KUKA KRL program: MyProgram_234().src

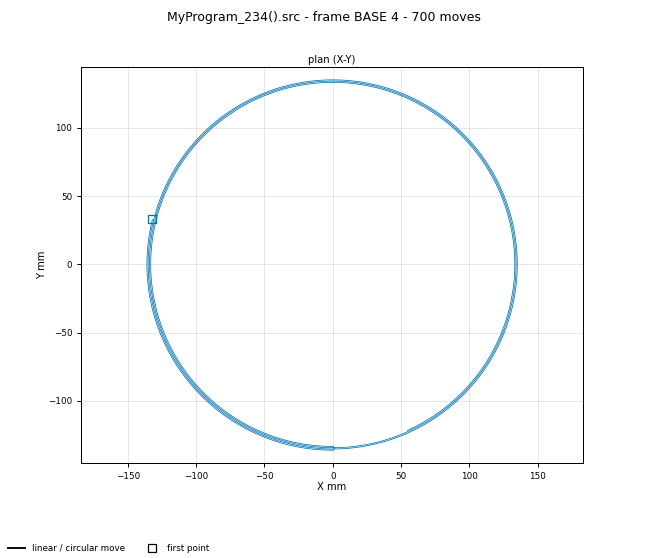
[picture p0: tool path of MyProgram_234().src in frame BASE 4, 700 of 700 moves have a stored position in this frame; points joined in program order, loops and branches not executed]
&ACCESS RVP
&REL 1
&PARAM TEMPLATE = C:\KRC\Roboter\Template\vorgabe
&PARAM EDITMASK = *
DEF MyProgram_234()
; ---- Setting reference (Base) ----
$BASE = BASE_DATA[4]

; --------------------------
; ---- Setting tool (TCP) ----
$TOOL = TOOL_DATA[3]
; --------------------------

$VEL.CP = VEL_APROX_PRINT
Startdeposition()
$VEL.CP = VEL_PRINT
LIN {X -132.079,Y 32.9632,Z 159,A 163.3178,B 23.9128,C -1.2869,E1 23.7896,E2 283.5753} C_DIS
LIN {X -133.2514,Y 27.8523,Z 159,A 165.544,B 23.9131,C -1.2806,E1 23.7882,E2 281.3509} C_DIS
LIN {X -134.047,Y 23.7201,Z 159,A 167.2359,B 23.9136,C -1.2711,E1 23.7874,E2 279.6721} C_DIS
LIN {X -134.6969,Y 19.7013,Z 159,A 168.9686,B 23.9138,C -1.2664,E1 23.7867,E2 277.9401} C_DIS
LIN {X -135.173,Y 16.1077,Z 159,A 170.4984,B 23.914,C -1.2616,E1 23.7861,E2 276.4127} C_DIS
LIN {X -135.6084,Y 11.907,Z 159,A 172.2964,B 23.9143,C -1.2567,E1 23.7857,E2 274.6154} C_DIS
LIN {X -135.8889,Y 8.0937,Z 159,A 173.8881,B 23.9146,C -1.2506,E1 23.7854,E2 273.0289} C_DIS
LIN {X -136.071,Y 3.9947,Z 159,A 175.6367,B 23.9148,C -1.246,E1 23.7852,E2 271.2807} C_DIS
LIN {X -136.1316,Y 0.0516,Z 159,A 177.3098,B 23.9151,C -1.2411,E1 23.7852,E2 269.609} C_DIS
LIN {X -136.08,Y -3.6704,Z 159,A 178.9234,B 23.9151,C -1.2383,E1 23.7852,E2 267.9922} C_DIS
LIN {X -135.9057,Y -7.8204,Z 159,A -179.3031,B 23.9154,C -1.2338,E1 23.7855,E2 266.2187} C_DIS
LIN {X -135.6203,Y -11.7657,Z 159,A -177.6067,B 23.9156,C -1.2299,E1 23.7859,E2 264.5213} C_DIS
LIN {X -135.25,Y -15.4619,Z 159,A -176.0236,B 23.9158,C -1.2258,E1 23.7863,E2 262.9385} C_DIS
LIN {X -134.7524,Y -19.3124,Z 159,A -174.416,B 23.9161,C -1.2192,E1 23.787,E2 261.337} C_DIS
LIN {X -133.9612,Y -24.1999,Z 159,A -171.5444,B 23.9146,C -1.2507,E1 23.7884,E2 258.3695} C_DIS
LIN {X -132.7292,Y -30.2346,Z 159,A -169.7414,B 23.9168,C -1.2043,E1 23.7894,E2 256.6705} C_DIS
LIN {X -131.8389,Y -33.9095,Z 159,A -168.2744,B 23.9173,C -1.1933,E1 23.7904,E2 255.2218} C_DIS
LIN {X -130.8523,Y -37.5362,Z 159,A -166.5488,B 23.9173,C -1.1953,E1 23.7917,E2 253.4807} C_DIS
LIN {X -129.8374,Y -40.9106,Z 159,A -165.065,B 23.9175,C -1.1908,E1 23.7929,E2 251.9992} C_DIS
LIN {X -128.7798,Y -44.1262,Z 159,A -163.6167,B 23.9176,C -1.1876,E1 23.7942,E2 250.5501} C_DIS
LIN {X -127.6866,Y -47.1974,Z 159,A -162.2254,B 23.9178,C -1.1844,E1 23.7955,E2 249.1585} C_DIS
LIN {X -126.4518,Y -50.4114,Z 159,A -160.7598,B 23.9179,C -1.1808,E1 23.797,E2 247.693} C_DIS
LIN {X -125.049,Y -53.7951,Z 159,A -159.4632,B 23.9187,C -1.1645,E1 23.7984,E2 246.4294} C_DIS
LIN {X -123.7178,Y -56.7903,Z 159,A -157.1398,B 23.9167,C -1.2064,E1 23.8013,E2 243.9887} C_DIS
LIN {X -121.2923,Y -61.8002,Z 159,A -155.5783,B 23.9188,C -1.1616,E1 23.8031,E2 242.5295} C_DIS
LIN {X -119.8894,Y -64.4838,Z 159,A -154.1181,B 23.9186,C -1.167,E1 23.805,E2 241.0477} C_DIS
LIN {X -117.6694,Y -68.4517,Z 159,A -152.2675,B 23.9189,C -1.1587,E1 23.8076,E2 239.2075} C_DIS
LIN {X -115.4192,Y -72.1811,Z 159,A -150.4067,B 23.9191,C -1.1551,E1 23.8103,E2 237.3456} C_DIS
LIN {X -113.1889,Y -75.6301,Z 159,A -148.648,B 23.9192,C -1.1521,E1 23.813,E2 235.5853} C_DIS
LIN {X -110.6731,Y -79.266,Z 159,A -146.7601,B 23.9194,C -1.1486,E1 23.816,E2 233.6961} C_DIS
LIN {X -107.9492,Y -82.9378,Z 159,A -144.8663,B 23.9197,C -1.1423,E1 23.8192,E2 231.8084} C_DIS
LIN {X -105.2261,Y -86.3665,Z 159,A -143.017,B 23.9199,C -1.1382,E1 23.8224,E2 229.9603} C_DIS
LIN {X -101.84,Y -90.3343,Z 159,A -140.897,B 23.9203,C -1.1294,E1 23.8263,E2 227.8521} C_DIS
LIN {X -99.3816,Y -93.0324,Z 159,A -139.2141,B 23.9201,C -1.1331,E1 23.8295,E2 226.1522} C_DIS
LIN {X -96.907,Y -95.6073,Z 159,A -137.545,B 23.9199,C -1.138,E1 23.8328,E2 224.4634} C_DIS
LIN {X -92.9629,Y -99.4464,Z 159,A -135.351,B 23.9204,C -1.127,E1 23.8372,E2 222.287} C_DIS
LIN {X -89.9747,Y -102.157,Z 159,A -133.0559,B 23.9192,C -1.1534,E1 23.8422,E2 219.9171} C_DIS
LIN {X -85.7356,Y -105.741,Z 159,A -131.3189,B 23.9207,C -1.1189,E1 23.8458,E2 218.2586} C_DIS
LIN {X -82.7538,Y -108.0899,Z 159,A -129.715,B 23.9208,C -1.1163,E1 23.8493,E2 216.655} C_DIS
LIN {X -79.0794,Y -110.8065,Z 159,A -127.8281,B 23.9211,C -1.1111,E1 23.8535,E2 214.774} C_DIS
LIN {X -75.5469,Y -113.2444,Z 159,A -126.0361,B 23.9212,C -1.1074,E1 23.8577,E2 212.9849} C_DIS
LIN {X -72.6974,Y -115.0944,Z 159,A -124.2034,B 23.9204,C -1.1254,E1 23.8621,E2 211.1015} C_DIS
LIN {X -69.2355,Y -117.21,Z 159,A -122.8138,B 23.9213,C -1.1068,E1 23.8654,E2 209.7535} C_DIS
LIN {X -66.0235,Y -119.0485,Z 159,A -121.2797,B 23.9214,C -1.1035,E1 23.8691,E2 208.223} C_DIS
LIN {X -62.1027,Y -121.1383,Z 159,A -119.4931,B 23.9217,C -1.0968,E1 23.8735,E2 206.4477} C_DIS
LIN {X -59.0691,Y -122.6463,Z 159,A -118.0743,B 23.9217,C -1.0947,E1 23.877,E2 205.0303} C_DIS
LIN {X -52.286,Y -125.6874,Z 159,A -114.8574,B 23.9217,C -1.0956,E1 23.8853,E2 201.8031} C_DIS
LIN {X -47.9859,Y -127.3913,Z 159,A -112.8439,B 23.9217,C -1.097,E1 23.8905,E2 199.7815} C_DIS
LIN {X -43.4345,Y -129.0146,Z 159,A -110.8603,B 23.9219,C -1.0927,E1 23.8958,E2 197.8045} C_DIS
LIN {X -39.8208,Y -130.1746,Z 159,A -109.3213,B 23.922,C -1.0885,E1 23.8998,E2 196.273} C_DIS
LIN {X -36.6839,Y -131.0932,Z 159,A -107.9375,B 23.922,C -1.088,E1 23.9036,E2 194.8882} C_DIS
LIN {X -32.9741,Y -132.0762,Z 159,A -106.2345,B 23.922,C -1.0915,E1 23.9082,E2 193.174} C_DIS
LIN {X -28.9465,Y -133.0162,Z 159,A -104.5737,B 23.9221,C -1.0865,E1 23.9127,E2 191.5233} C_DIS
LIN {X -25.5638,Y -133.7074,Z 159,A -103.1858,B 23.9223,C -1.0826,E1 23.9165,E2 190.1435} C_DIS
LIN {X -20.5942,Y -134.5627,Z 159,A -100.9853,B 23.9222,C -1.0859,E1 23.9226,E2 187.9326} C_DIS
LIN {X -16.4484,Y -135.1324,Z 159,A -98.8515,B 23.9213,C -1.1049,E1 23.9286,E2 185.7503} C_DIS
LIN {X -12.5936,Y -135.5462,Z 159,A -96.9315,B 23.9207,C -1.1198,E1 23.9341,E2 183.7925} C_DIS
LIN {X -7.2101,Y -135.9389,Z 159,A -95.2727,B 23.9221,C -1.0878,E1 23.9385,E2 182.212} C_DIS
LIN {X 0.5173,Y -136.1287,Z 159,A -91.6014,B 23.9211,C -1.1103,E1 23.9489,E2 178.4853} C_DIS
LIN {X 0.5173,Y -136.1287,Z 159,A -91.6014,B 23.9211,C -1.1103,E1 23.9489,E2 178.4853} C_DIS
Enddeposition()
LIN {X 0.9368,Y -135.1941,Z 159,A -91.8649,B 22.4196,C -0.8172,E1 22.4349,E2 179.316} C_DIS
Startdeposition()
$VEL.CP = VEL_PRINT
LIN {X -3.0281,Y -135.1695,Z 159,A -93.7042,B 22.4199,C -0.8092,E1 22.4297,E2 181.1764} C_DIS
LIN {X -7.7949,Y -134.9776,Z 159,A -95.9195,B 22.4202,C -0.7999,E1 22.4234,E2 183.4167} C_DIS
LIN {X -13.0956,Y -134.5658,Z 159,A -98.0516,B 22.42,C -0.8058,E1 22.4175,E2 185.5345} C_DIS
LIN {X -16.1305,Y -134.2357,Z 159,A -99.3289,B 22.42,C -0.8068,E1 22.414,E2 186.8101} C_DIS
LIN {X -19.4901,Y -133.7897,Z 159,A -100.8591,B 22.42,C -0.8027,E1 22.4097,E2 188.3524} C_DIS
LIN {X -23.6224,Y -133.1218,Z 159,A -102.3216,B 22.4196,C -0.8179,E1 22.4058,E2 189.7764} C_DIS
LIN {X -26.7677,Y -132.5251,Z 159,A -103.9188,B 22.4199,C -0.8072,E1 22.4014,E2 191.4039} C_DIS
LIN {X -30.2748,Y -131.7681,Z 159,A -105.4244,B 22.4199,C -0.8086,E1 22.3973,E2 192.9078} C_DIS
LIN {X -33.5797,Y -130.9652,Z 159,A -106.8089,B 22.4198,C -0.8121,E1 22.3935,E2 194.2854} C_DIS
LIN {X -36.6063,Y -130.1514,Z 159,A -108.1864,B 22.4198,C -0.8107,E1 22.3898,E2 195.669} C_DIS
LIN {X -39.882,Y -129.1855,Z 159,A -109.6302,B 22.4198,C -0.8119,E1 22.3859,E2 197.1124} C_DIS
LIN {X -43.3138,Y -128.0767,Z 159,A -111.3197,B 22.42,C -0.8056,E1 22.3814,E2 198.8218} C_DIS
LIN {X -47.6534,Y -126.5249,Z 159,A -113.1109,B 22.4197,C -0.8149,E1 22.3768,E2 200.5927} C_DIS
LIN {X -50.6546,Y -125.3533,Z 159,A -114.5476,B 22.4197,C -0.813,E1 22.373,E2 202.038} C_DIS
LIN {X -54.6129,Y -123.6817,Z 159,A -116.7429,B 22.4203,C -0.7977,E1 22.3673,E2 204.2792} C_DIS
LIN {X -58.0744,Y -122.0931,Z 159,A -117.7099,B 22.4192,C -0.8294,E1 22.365,E2 205.1657} C_DIS
LIN {X -62.044,Y -120.1269,Z 159,A -119.8272,B 22.4195,C -0.8207,E1 22.3597,E2 207.3123} C_DIS
LIN {X -64.6397,Y -118.75,Z 159,A -121.1817,B 22.4195,C -0.8173,E1 22.3563,E2 208.6799} C_DIS
LIN {X -68.3399,Y -116.6599,Z 159,A -123.4642,B 22.4203,C -0.798,E1 22.3507,E2 211.0209} C_DIS
LIN {X -72.4236,Y -114.1698,Z 159,A -124.6995,B 22.4189,C -0.8371,E1 22.348,E2 212.1577} C_DIS
LIN {X -76.606,Y -111.4063,Z 159,A -127.1393,B 22.4193,C -0.8262,E1 22.3422,E2 214.6355} C_DIS
LIN {X -80.2636,Y -108.801,Z 159,A -129.009,B 22.4191,C -0.831,E1 22.338,E2 216.4999} C_DIS
LIN {X -83.739,Y -106.1494,Z 159,A -130.9102,B 22.4191,C -0.8321,E1 22.3338,E2 218.4059} C_DIS
LIN {X -87.1969,Y -103.3281,Z 159,A -133.1146,B 22.4194,C -0.8216,E1 22.329,E2 220.6475} C_DIS
LIN {X -90.0311,Y -100.8676,Z 159,A -134.0842,B 22.4183,C -0.8528,E1 22.3271,E2 221.5394} C_DIS
LIN {X -93.7404,Y -97.4307,Z 159,A -136.5561,B 22.4187,C -0.8423,E1 22.322,E2 224.0503} C_DIS
LIN {X -96.7962,Y -94.3953,Z 159,A -138.4289,B 22.4187,C -0.8441,E1 22.3183,E2 225.9274} C_DIS
LIN {X -99.8464,Y -91.1631,Z 159,A -140.1658,B 22.4183,C -0.8548,E1 22.315,E2 227.6446} C_DIS
LIN {X -102.1643,Y -88.5577,Z 159,A -141.8369,B 22.4185,C -0.8496,E1 22.3119,E2 229.338} C_DIS
LIN {X -105.1304,Y -85.0145,Z 159,A -143.761,B 22.4182,C -0.8557,E1 22.3085,E2 231.256} C_DIS
LIN {X -108.0038,Y -81.3329,Z 159,A -145.7259,B 22.418,C -0.8612,E1 22.3052,E2 233.217} C_DIS
LIN {X -110.675,Y -77.6594,Z 159,A -147.7071,B 22.418,C -0.8635,E1 22.3019,E2 235.2031} C_DIS
LIN {X -113.2164,Y -73.9053,Z 159,A -149.6464,B 22.4178,C -0.8677,E1 22.2989,E2 237.1425} C_DIS
LIN {X -115.5116,Y -70.2641,Z 159,A -151.4667,B 22.4176,C -0.8726,E1 22.2963,E2 238.9601} C_DIS
LIN {X -117.7755,Y -66.3988,Z 159,A -153.3603,B 22.4174,C -0.878,E1 22.2936,E2 240.8508} C_DIS
LIN {X -119.7044,Y -62.8503,Z 159,A -155.0786,B 22.4173,C -0.8824,E1 22.2914,E2 242.5677} C_DIS
LIN {X -121.6017,Y -59.1012,Z 159,A -156.7614,B 22.4169,C -0.8917,E1 22.2893,E2 244.2362} C_DIS
LIN {X -123.8092,Y -54.3244,Z 159,A -158.9741,B 22.4166,C -0.8988,E1 22.2868,E2 246.4438} C_DIS
LIN {X -124.9315,Y -51.688,Z 159,A -160.3608,B 22.4168,C -0.8947,E1 22.2852,E2 247.8499} C_DIS
LIN {X -126.5688,Y -47.5361,Z 159,A -162.2011,B 22.4165,C -0.9026,E1 22.2834,E2 249.6814} C_DIS
LIN {X -127.8142,Y -44.0784,Z 159,A -163.722,B 22.4163,C -0.9088,E1 22.282,E2 251.1955} C_DIS
LIN {X -129.0675,Y -40.2673,Z 159,A -165.3832,B 22.416,C -0.9156,E1 22.2806,E2 252.8496} C_DIS
LIN {X -130.0053,Y -37.1251,Z 159,A -167.1173,B 22.4164,C -0.9048,E1 22.2792,E2 254.6235} C_DIS
LIN {X -130.8711,Y -33.9505,Z 159,A -168.4639,B 22.4162,C -0.9111,E1 22.2783,E2 255.9622} C_DIS
LIN {X -133.1369,Y -23.5378,Z 159,A -172.7695,B 22.4153,C -0.9344,E1 22.2758,E2 260.2352} C_DIS
LIN {X -133.6941,Y -20.1397,Z 159,A -174.3597,B 22.4153,C -0.9332,E1 22.2751,E2 261.8391} C_DIS
LIN {X -134.2618,Y -15.912,Z 159,A -176.0343,B 22.4148,C -0.9448,E1 22.2745,E2 263.4945} C_DIS
LIN {X -134.6144,Y -12.5897,Z 159,A -177.5154,B 22.4148,C -0.9465,E1 22.2741,E2 264.9812} C_DIS
LIN {X -134.9389,Y -8.4233,Z 159,A -179.2792,B 22.4145,C -0.9524,E1 22.2738,E2 266.7412} C_DIS
LIN {X -135.11,Y -4.9807,Z 159,A 179.14,B 22.4145,C -0.9519,E1 22.2736,E2 268.3341} C_DIS
LIN {X -135.1996,Y -0.8442,Z 159,A 177.4322,B 22.4142,C -0.9595,E1 22.2736,E2 270.0335} C_DIS
LIN {X -135.1606,Y 3.3519,Z 159,A 175.6326,B 22.4141,C -0.9643,E1 22.2736,E2 271.8327} C_DIS
LIN {X -135.0229,Y 6.949,Z 159,A 174.1184,B 22.4138,C -0.9698,E1 22.2738,E2 273.3427} C_DIS
LIN {X -134.735,Y 11.2223,Z 159,A 172.2572,B 22.4137,C -0.9736,E1 22.2742,E2 275.2065} C_DIS
LIN {X -134.2965,Y 15.6212,Z 159,A 170.3647,B 22.4135,C -0.9788,E1 22.2747,E2 277.0981} C_DIS
LIN {X -133.7907,Y 19.4832,Z 159,A 168.7199,B 22.4132,C -0.9844,E1 22.2754,E2 278.7393} C_DIS
LIN {X -133.0853,Y 23.8263,Z 159,A 166.925,B 22.4128,C -0.9934,E1 22.2762,E2 280.5223} C_DIS
LIN {X -132.4612,Y 27.0816,Z 159,A 165.4622,B 22.4128,C -0.9954,E1 22.277,E2 281.9897} C_DIS
LIN {X -131.5133,Y 31.3644,Z 159,A 163.8004,B 22.4121,C -1.0099,E1 22.278,E2 283.6244} C_DIS
LIN {X -130.7732,Y 34.3223,Z 159,A 161.9635,B 22.413,C -0.9903,E1 22.2793,E2 285.525} C_DIS
LIN {X -129.8613,Y 37.6236,Z 159,A 161.0027,B 22.4119,C -1.0162,E1 22.28,E2 286.4239} C_DIS
LIN {X -128.0076,Y 43.5208,Z 159,A 158.2134,B 22.4119,C -1.0169,E1 22.2824,E2 289.2292} C_DIS
LIN {X -126.5522,Y 47.5804,Z 159,A 156.3461,B 22.4117,C -1.0209,E1 22.2842,E2 291.098} C_DIS
LIN {X -125.2287,Y 50.9637,Z 159,A 154.8328,B 22.4114,C -1.0267,E1 22.2857,E2 292.6055} C_DIS
LIN {X -123.992,Y 53.9014,Z 159,A 153.4528,B 22.4113,C -1.0295,E1 22.2872,E2 293.9866} C_DIS
LIN {X -122.6155,Y 56.9631,Z 159,A 152.0207,B 22.4111,C -1.0334,E1 22.2889,E2 295.4174} C_DIS
LIN {X -121.1128,Y 60.0924,Z 159,A 150.5165,B 22.4111,C -1.0363,E1 22.2907,E2 296.9231} C_DIS
LIN {X -119.2292,Y 63.752,Z 159,A 148.7776,B 22.4108,C -1.0417,E1 22.293,E2 298.6583} C_DIS
LIN {X -117.2847,Y 67.2624,Z 159,A 146.9782,B 22.4108,C -1.0423,E1 22.2955,E2 300.4667} C_DIS
LIN {X -115.0045,Y 71.0913,Z 159,A 145.0611,B 22.4106,C -1.0464,E1 22.2982,E2 302.3841} C_DIS
LIN {X -112.9386,Y 74.3283,Z 159,A 143.4277,B 22.4104,C -1.0507,E1 22.3007,E2 304.0154} C_DIS
LIN {X -110.4125,Y 78.0316,Z 159,A 141.5521,B 22.4101,C -1.057,E1 22.3037,E2 305.885} C_DIS
LIN {X -107.8054,Y 81.5957,Z 159,A 139.556,B 22.4101,C -1.0566,E1 22.307,E2 307.893} C_DIS
LIN {X -105.1746,Y 84.9597,Z 159,A 137.7114,B 22.41,C -1.0598,E1 22.3103,E2 309.7389} C_DIS
LIN {X -99.9633,Y 91.0343,Z 159,A 134.2089,B 22.4098,C -1.0636,E1 22.3167,E2 313.2494} C_DIS
LIN {X -96.201,Y 95.002,Z 159,A 132.0334,B 22.4093,C -1.0754,E1 22.3209,E2 315.4042} C_DIS
LIN {X -92.9702,Y 98.1654,Z 159,A 130.1303,B 22.409,C -1.0805,E1 22.3247,E2 317.3027} C_DIS
LIN {X -89.188,Y 101.6136,Z 159,A 128.0456,B 22.4086,C -1.0892,E1 22.329,E2 319.3739} C_DIS
LIN {X -86.0424,Y 104.291,Z 159,A 125.762,B 22.4095,C -1.0695,E1 22.3341,E2 321.7192} C_DIS
LIN {X -82.4871,Y 107.1256,Z 159,A 123.8971,B 22.4092,C -1.0763,E1 22.3382,E2 323.5739} C_DIS
LIN {X -79.195,Y 109.5811,Z 159,A 122.5954,B 22.4082,C -1.0993,E1 22.341,E2 324.8203} C_DIS
LIN {X -75.9198,Y 111.8751,Z 159,A 120.835,B 22.4082,C -1.0997,E1 22.345,E2 326.5864} C_DIS
LIN {X -69.1781,Y 116.1647,Z 159,A 117.6362,B 22.4075,C -1.1144,E1 22.3525,E2 329.758} C_DIS
LIN {X -66.4481,Y 117.7478,Z 159,A 116.055,B 22.4079,C -1.1058,E1 22.3564,E2 331.3671} C_DIS
LIN {X -62.7463,Y 119.759,Z 159,A 114.3724,B 22.4075,C -1.1134,E1 22.3605,E2 333.0349} C_DIS
LIN {X -59.6838,Y 121.3143,Z 159,A 112.8999,B 22.4075,C -1.115,E1 22.3642,E2 334.5078} C_DIS
LIN {X -56.5735,Y 122.7957,Z 159,A 111.4519,B 22.4073,C -1.1177,E1 22.3679,E2 335.9526} C_DIS
LIN {X -53.5676,Y 124.1363,Z 159,A 110.0567,B 22.4072,C -1.1197,E1 22.3714,E2 337.3462} C_DIS
LIN {X -50.4397,Y 125.4399,Z 159,A 108.5749,B 22.4072,C -1.1197,E1 22.3753,E2 338.8321} C_DIS
LIN {X -47.2933,Y 126.6597,Z 159,A 107.1857,B 22.407,C -1.1234,E1 22.3789,E2 340.2148} C_DIS
LIN {X -43.6108,Y 127.9763,Z 159,A 105.4395,B 22.4071,C -1.1213,E1 22.3835,E2 341.9702} C_DIS
LIN {X -40.2541,Y 129.0716,Z 159,A 103.4149,B 22.4082,C -1.0991,E1 22.3891,E2 344.0571} C_DIS
LIN {X -35.59,Y 130.4351,Z 159,A 101.9715,B 22.4067,C -1.1292,E1 22.3927,E2 345.4241} C_DIS
LIN {X -31.6897,Y 131.4349,Z 159,A 100.2111,B 22.4067,C -1.1283,E1 22.3975,E2 347.1896} C_DIS
LIN {X -28.2315,Y 132.2212,Z 159,A 98.7141,B 22.4067,C -1.1299,E1 22.4016,E2 348.6845} C_DIS
LIN {X -24.8067,Y 132.9073,Z 159,A 97.2744,B 22.4066,C -1.1329,E1 22.4055,E2 350.1182} C_DIS
LIN {X -22.2073,Y 133.365,Z 159,A 96.1246,B 22.4066,C -1.1323,E1 22.4087,E2 351.2708} C_DIS
LIN {X -18.7934,Y 133.8892,Z 159,A 94.6393,B 22.4066,C -1.1322,E1 22.4128,E2 352.7577} C_DIS
LIN {X -14.6909,Y 134.4011,Z 159,A 92.8678,B 22.4066,C -1.1322,E1 22.4177,E2 354.5303} C_DIS
LIN {X -10.9753,Y 134.7558,Z 159,A 91.2739,B 22.4066,C -1.1324,E1 22.4222,E2 356.1248} C_DIS
LIN {X -6.8495,Y 135.0279,Z 159,A 89.5555,B 22.4065,C -1.1346,E1 22.4269,E2 357.838} C_DIS
LIN {X -2.9332,Y 135.1715,Z 159,A 87.7203,B 22.4069,C -1.1269,E1 22.4321,E2 359.6935} C_DIS
LIN {X 1.7244,Y 135.1916,Z 159,A 85.8443,B 22.4066,C -1.1318,E1 22.4373,E2 361.5567} C_DIS
LIN {X 6.0742,Y 135.0666,Z 159,A 84.1504,B 22.4063,C -1.1389,E1 22.442,E2 363.2314} C_DIS
LIN {X 9.5609,Y 134.8633,Z 159,A 82.5125,B 22.4066,C -1.1315,E1 22.4466,E2 364.888} C_DIS
LIN {X 12.873,Y 134.5872,Z 159,A 81.2086,B 22.4064,C -1.1362,E1 22.4502,E2 366.1787} C_DIS
LIN {X 16.2698,Y 134.2191,Z 159,A 79.8009,B 22.4064,C -1.1378,E1 22.4541,E2 367.581} C_DIS
LIN {X 19.2971,Y 133.8173,Z 159,A 78.456,B 22.4064,C -1.1351,E1 22.4578,E2 368.9317} C_DIS
LIN {X 23.082,Y 133.2185,Z 159,A 76.7148,B 22.4068,C -1.129,E1 22.4627,E2 370.687} C_DIS
LIN {X 26.9196,Y 132.4942,Z 159,A 75.1512,B 22.4066,C -1.1326,E1 22.4669,E2 372.2391} C_DIS
LIN {X 30.3615,Y 131.7483,Z 159,A 73.7166,B 22.4065,C -1.1345,E1 22.4708,E2 373.6665} C_DIS
LIN {X 33.361,Y 131.0207,Z 159,A 72.3996,B 22.4065,C -1.1333,E1 22.4744,E2 374.9844} C_DIS
LIN {X 36.6495,Y 130.1393,Z 159,A 70.8758,B 22.4068,C -1.1284,E1 22.4785,E2 376.5181} C_DIS
LIN {X 40.6368,Y 128.9507,Z 159,A 69.0872,B 22.4069,C -1.1258,E1 22.4833,E2 378.3098} C_DIS
LIN {X 44.6491,Y 127.6164,Z 159,A 67.4221,B 22.4067,C -1.1303,E1 22.4876,E2 379.9595} C_DIS
LIN {X 47.6399,Y 126.5299,Z 159,A 66.0249,B 22.4069,C -1.1267,E1 22.4913,E2 381.3629} C_DIS
LIN {X 51.3043,Y 125.0914,Z 159,A 63.9617,B 22.4078,C -1.1061,E1 22.4968,E2 383.4748} C_DIS
LIN {X 54.8227,Y 123.5878,Z 159,A 62.9325,B 22.4066,C -1.1326,E1 22.4992,E2 384.4317} C_DIS
LIN {X 58.4531,Y 121.9122,Z 159,A 61.0267,B 22.4072,C -1.1204,E1 22.5041,E2 386.3639} C_DIS
LIN {X 61.5059,Y 120.4008,Z 159,A 59.6207,B 22.4072,C -1.1204,E1 22.5076,E2 387.7658} C_DIS
LIN {X 64.8255,Y 118.6486,Z 159,A 57.9575,B 22.4074,C -1.1146,E1 22.5117,E2 389.4386} C_DIS
LIN {X 68.9881,Y 116.2779,Z 159,A 56.0845,B 22.4072,C -1.1192,E1 22.5162,E2 391.2931} C_DIS
LIN {X 72.1374,Y 114.3505,Z 159,A 54.384,B 22.4076,C -1.1102,E1 22.5203,E2 393.011} C_DIS
LIN {X 75.9628,Y 111.846,Z 159,A 52.4437,B 22.4078,C -1.1069,E1 22.5248,E2 394.9527} C_DIS
LIN {X 79.7313,Y 109.1921,Z 159,A 50.7695,B 22.4073,C -1.1171,E1 22.5285,E2 396.5936} C_DIS
LIN {X 82.2309,Y 107.3216,Z 159,A 49.2041,B 22.408,C -1.1029,E1 22.5321,E2 398.1898} C_DIS
LIN {X 88.037,Y 102.6128,Z 159,A 46.3472,B 22.4076,C -1.1121,E1 22.5382,E2 401.0104} C_DIS
LIN {X 91.784,Y 99.2758,Z 159,A 43.5996,B 22.4092,C -1.0773,E1 22.544,E2 403.8364} C_DIS
LIN {X 94.5699,Y 96.625,Z 159,A 42.4795,B 22.4082,C -1.0988,E1 22.5462,E2 404.895} C_DIS
LIN {X 97.0015,Y 94.1837,Z 159,A 40.8398,B 22.4087,C -1.0868,E1 22.5494,E2 406.5582} C_DIS
LIN {X 101.5471,Y 89.2646,Z 159,A 38.0984,B 22.4088,C -1.0851,E1 22.5546,E2 409.2903} C_DIS
LIN {X 104.2107,Y 86.1392,Z 159,A 36.2924,B 22.4091,C -1.0778,E1 22.5578,E2 411.1061} C_DIS
LIN {X 106.888,Y 82.7936,Z 159,A 34.6906,B 22.4089,C -1.084,E1 22.5606,E2 412.6832} C_DIS
LIN {X 108.9438,Y 80.0692,Z 159,A 33.0648,B 22.4094,C -1.0715,E1 22.5633,E2 414.3329} C_DIS
LIN {X 113.1652,Y 73.9842,Z 159,A 30.1744,B 22.4092,C -1.0758,E1 22.5678,E2 417.196} C_DIS
LIN {X 115.8094,Y 69.7716,Z 159,A 27.8306,B 22.41,C -1.0584,E1 22.5713,E2 419.5716} C_DIS
LIN {X 118.0359,Y 65.9355,Z 159,A 25.9583,B 22.4102,C -1.0537,E1 22.5739,E2 421.4453} C_DIS
LIN {X 120.3389,Y 61.6275,Z 159,A 23.4907,B 22.4114,C -1.0282,E1 22.5772,E2 423.9647} C_DIS
LIN {X 122.3288,Y 57.5811,Z 159,A 22.1085,B 22.4104,C -1.0491,E1 22.5788,E2 425.284} C_DIS
LIN {X 123.7306,Y 54.5034,Z 159,A 20.5324,B 22.4109,C -1.0378,E1 22.5806,E2 426.8798} C_DIS
LIN {X 125.3191,Y 50.7395,Z 159,A 18.8865,B 22.4109,C -1.0371,E1 22.5823,E2 428.5174} C_DIS
LIN {X 126.7332,Y 47.0971,Z 159,A 17.2464,B 22.4111,C -1.033,E1 22.5839,E2 430.1579} C_DIS
LIN {X 128.0311,Y 43.4461,Z 159,A 15.7569,B 22.4111,C -1.0357,E1 22.5853,E2 431.6308} C_DIS
LIN {X 129.1404,Y 40.0291,Z 159,A 13.9777,B 22.4118,C -1.0182,E1 22.5868,E2 433.4443} C_DIS
LIN {X 130.2027,Y 36.4226,Z 159,A 12.5724,B 22.4116,C -1.0228,E1 22.5879,E2 434.8284} C_DIS
LIN {X 131.1083,Y 33.0157,Z 159,A 11.0714,B 22.4118,C -1.0178,E1 22.5889,E2 436.3326} C_DIS
LIN {X 132.1173,Y 28.7128,Z 159,A 9.2185,B 22.412,C -1.013,E1 22.5901,E2 438.1859} C_DIS
LIN {X 132.8234,Y 25.2458,Z 159,A 7.7394,B 22.4122,C -1.0094,E1 22.5909,E2 439.6648} C_DIS
LIN {X 133.5538,Y 21.0452,Z 159,A 5.9287,B 22.4124,C -1.0035,E1 22.5917,E2 441.4789} C_DIS
LIN {X 134.0729,Y 17.4323,Z 159,A 4.4016,B 22.4126,C -0.9996,E1 22.5923,E2 443.006} C_DIS
LIN {X 134.5545,Y 13.214,Z 159,A 2.6198,B 22.4128,C -0.9947,E1 22.5928,E2 444.7886} C_DIS
LIN {X 134.848,Y 9.7697,Z 159,A 1.1421,B 22.413,C -0.9893,E1 22.5932,E2 446.2703} C_DIS
LIN {X 135.0997,Y 5.2451,Z 159,A -0.737,B 22.4132,C -0.9853,E1 22.5934,E2 448.1474} C_DIS
LIN {X 135.1968,Y 1.2733,Z 159,A -2.4429,B 22.4135,C -0.9787,E1 22.5935,E2 449.8591} C_DIS
LIN {X 135.1333,Y -4.3323,Z 159,A -4.6723,B 22.4135,C -0.9784,E1 22.5935,E2 452.0743} C_DIS
LIN {X 134.9023,Y -9.0163,Z 159,A -6.8563,B 22.4141,C -0.962,E1 22.5931,E2 454.2864} C_DIS
LIN {X 134.5838,Y -12.9088,Z 159,A -8.3855,B 22.4141,C -0.963,E1 22.5927,E2 455.8026} C_DIS
LIN {X 134.1542,Y -16.8121,Z 159,A -10.1901,B 22.4146,C -0.9505,E1 22.5921,E2 457.6277} C_DIS
LIN {X 133.5459,Y -21.0965,Z 159,A -11.8162,B 22.4144,C -0.9552,E1 22.5914,E2 459.231} C_DIS
LIN {X 132.9134,Y -24.7749,Z 159,A -13.5155,B 22.4149,C -0.9441,E1 22.5906,E2 460.9479} C_DIS
LIN {X 132.1727,Y -28.4561,Z 159,A -14.9901,B 22.4149,C -0.9449,E1 22.5897,E2 462.4106} C_DIS
LIN {X 131.4151,Y -31.7719,Z 159,A -16.4018,B 22.4149,C -0.9418,E1 22.5888,E2 463.8211} C_DIS
LIN {X 130.6037,Y -34.9577,Z 159,A -17.7992,B 22.4151,C -0.9372,E1 22.5879,E2 465.2215} C_DIS
LIN {X 129.6561,Y -38.3244,Z 159,A -19.2823,B 22.4153,C -0.9325,E1 22.5867,E2 466.7074} C_DIS
LIN {X 128.047,Y -43.4031,Z 159,A -21.665,B 22.4159,C -0.919,E1 22.5846,E2 469.1099} C_DIS
LIN {X 126.6353,Y -47.3585,Z 159,A -23.361,B 22.4159,C -0.9178,E1 22.583,E2 470.7985} C_DIS
LIN {X 125.048,Y -51.4081,Z 159,A -25.4175,B 22.4165,C -0.9013,E1 22.5808,E2 472.885} C_DIS
LIN {X 123.7289,Y -54.5073,Z 159,A -26.4957,B 22.416,C -0.9146,E1 22.5797,E2 473.9219} C_DIS
LIN {X 122.5747,Y -57.0514,Z 159,A -27.704,B 22.4162,C -0.9098,E1 22.5783,E2 475.1353} C_DIS
LIN {X 121.0784,Y -60.1621,Z 159,A -29.2463,B 22.4165,C -0.9014,E1 22.5764,E2 476.6902} C_DIS
LIN {X 119.2725,Y -63.6714,Z 159,A -30.9294,B 22.4167,C -0.8959,E1 22.5742,E2 478.3775} C_DIS
LIN {X 117.1423,Y -67.5099,Z 159,A -32.766,B 22.4169,C -0.8917,E1 22.5716,E2 480.2144} C_DIS
LIN {X 114.9924,Y -71.1106,Z 159,A -34.8694,B 22.4177,C -0.8702,E1 22.5685,E2 482.3617} C_DIS
LIN {X 112.8317,Y -74.4907,Z 159,A -36.0037,B 22.4168,C -0.8939,E1 22.5669,E2 483.428} C_DIS
LIN {X 110.8692,Y -77.3815,Z 159,A -37.6618,B 22.4173,C -0.8808,E1 22.5642,E2 485.111} C_DIS
LIN {X 108.5569,Y -80.5932,Z 159,A -39.2925,B 22.4173,C -0.8786,E1 22.5615,E2 486.7386} C_DIS
LIN {X 106.2984,Y -83.5493,Z 159,A -40.9195,B 22.4176,C -0.8718,E1 22.5587,E2 488.3745} C_DIS
LIN {X 104.1689,Y -86.1897,Z 159,A -42.3372,B 22.4177,C -0.869,E1 22.5562,E2 489.7921} C_DIS
LIN {X 101.1842,Y -89.675,Z 159,A -44.2845,B 22.4179,C -0.8639,E1 22.5527,E2 491.7429} C_DIS
LIN {X 98.11,Y -93.0289,Z 159,A -46.3278,B 22.4183,C -0.8533,E1 22.5487,E2 493.8038} C_DIS
LIN {X 95.0539,Y -96.1494,Z 159,A -48.0288,B 22.4183,C -0.8562,E1 22.5454,E2 495.4889} C_DIS
LIN {X 92.1181,Y -98.965,Z 159,A -49.6416,B 22.4182,C -0.8577,E1 22.5422,E2 497.0903} C_DIS
LIN {X 89.2836,Y -101.5303,Z 159,A -51.6284,B 22.4189,C -0.8357,E1 22.5379,E2 499.1256} C_DIS
LIN {X 86.5324,Y -103.8852,Z 159,A -52.7912,B 22.4184,C -0.8508,E1 22.5355,E2 500.244} C_DIS
LIN {X 83.5495,Y -106.2982,Z 159,A -54.5109,B 22.4187,C -0.8426,E1 22.5317,E2 501.9779} C_DIS
LIN {X 80.2383,Y -108.8196,Z 159,A -56.2826,B 22.4189,C -0.8384,E1 22.5278,E2 503.7532} C_DIS
LIN {X 76.0222,Y -111.8058,Z 159,A -58.4754,B 22.419,C -0.8339,E1 22.5227,E2 505.9494} C_DIS
LIN {X 72.1447,Y -114.3459,Z 159,A -60.547,B 22.4193,C -0.8248,E1 22.5178,E2 508.0371} C_DIS
LIN {X 67.7844,Y -116.9834,Z 159,A -62.5338,B 22.4192,C -0.8294,E1 22.5131,E2 510.005} C_DIS
LIN {X 63.8333,Y -119.1855,Z 159,A -64.4254,B 22.4192,C -0.8273,E1 22.5085,E2 511.8958} C_DIS
LIN {X 60.7559,Y -120.7826,Z 159,A -66.0195,B 22.4195,C -0.8187,E1 22.5044,E2 513.5074} C_DIS
LIN {X 55.9191,Y -123.0974,Z 159,A -68.0671,B 22.4193,C -0.8262,E1 22.4993,E2 515.5295} C_DIS
LIN {X 53.3772,Y -124.2187,Z 159,A -69.2808,B 22.4194,C -0.8227,E1 22.4962,E2 516.749} C_DIS
LIN {X 49.9131,Y -125.6522,Z 159,A -70.8478,B 22.4194,C -0.8215,E1 22.4922,E2 518.3151} C_DIS
LIN {X 45.1673,Y -127.4354,Z 159,A -72.9768,B 22.4195,C -0.8196,E1 22.4866,E2 520.4439} C_DIS
LIN {X 41.318,Y -128.733,Z 159,A -74.8153,B 22.4198,C -0.8119,E1 22.4817,E2 522.2989} C_DIS
LIN {X 38.1483,Y -129.7077,Z 159,A -76.6306,B 22.4205,C -0.7904,E1 22.4767,E2 524.1667} C_DIS
LIN {X 33.7779,Y -130.9149,Z 159,A -77.9071,B 22.4195,C -0.8196,E1 22.4734,E2 525.3645} C_DIS
LIN {X 30.0108,Y -131.8284,Z 159,A -79.6847,B 22.4198,C -0.8115,E1 22.4686,E2 527.1604} C_DIS
LIN {X 26.1897,Y -132.6427,Z 159,A -81.4731,B 22.4201,C -0.8037,E1 22.4636,E2 528.9669} C_DIS
LIN {X 21.8875,Y -133.4184,Z 159,A -83.188,B 22.4199,C -0.8089,E1 22.4589,E2 530.666} C_DIS
LIN {X 17.7735,Y -134.0282,Z 159,A -85.0335,B 22.4201,C -0.8038,E1 22.4538,E2 532.5232} C_DIS
LIN {X 13.9227,Y -134.4837,Z 159,A -86.5019,B 22.4198,C -0.8112,E1 22.4498,E2 533.9709} C_DIS
LIN {X 10.6148,Y -134.7859,Z 159,A -87.9154,B 22.4198,C -0.8102,E1 22.4458,E2 535.3861} C_DIS
LIN {X 5.4273,Y -135.0926,Z 159,A -90.1899,B 22.42,C -0.806,E1 22.4395,E2 537.6708} C_DIS
LIN {X 1.8312,Y -135.1898,Z 159,A -91.8209,B 22.4202,C -0.8004,E1 22.4349,E2 539.316} C_DIS
LIN {X 1.8312,Y -135.1898,Z 159,A -91.8209,B 22.4202,C -0.8004,E1 22.4349,E2 539.316} C_DIS
Enddeposition()
LIN {X 0.9317,Y -134.2705,Z 159,A -91.4866,B 21.2937,C -0.6553,E1 21.3046,E2 539.2529} C_DIS
Startdeposition()
$VEL.CP = VEL_PRINT
LIN {X 4.7236,Y -134.1914,Z 159,A -89.4063,B 21.293,C -0.6767,E1 21.3106,E2 537.1142} C_DIS
LIN {X 8.0515,Y -134.0321,Z 159,A -88.0785,B 21.2931,C -0.673,E1 21.3142,E2 535.7972} C_DIS
LIN {X 12.0653,Y -133.7325,Z 159,A -86.3699,B 21.2931,C -0.6733,E1 21.319,E2 534.0887} C_DIS
LIN {X 15.6264,Y -133.3613,Z 159,A -84.9161,B 21.2932,C -0.6708,E1 21.323,E2 532.6431} C_DIS
LIN {X 18.7648,Y -132.9559,Z 159,A -83.4633,B 21.293,C -0.6763,E1 21.3271,E2 531.1765} C_DIS
LIN {X 22.0237,Y -132.4549,Z 159,A -82.2179,B 21.2932,C -0.6699,E1 21.3304,E2 529.9502} C_DIS
LIN {X 24.6854,Y -131.9858,Z 159,A -80.8414,B 21.2929,C -0.6811,E1 21.3343,E2 528.5449} C_DIS
LIN {X 28.1125,Y -131.2976,Z 159,A -79.5107,B 21.2931,C -0.6749,E1 21.3379,E2 527.2332} C_DIS
LIN {X 31.1798,Y -130.6033,Z 159,A -78.0774,B 21.2929,C -0.6804,E1 21.3418,E2 525.7873} C_DIS
LIN {X 34.0677,Y -129.8807,Z 159,A -76.9293,B 21.2931,C -0.676,E1 21.3449,E2 524.6534} C_DIS
LIN {X 36.9471,Y -129.0925,Z 159,A -75.5575,B 21.2929,C -0.6818,E1 21.3486,E2 523.2682} C_DIS
LIN {X 40.0776,Y -128.1551,Z 159,A -74.1648,B 21.2929,C -0.6833,E1 21.3523,E2 521.8744} C_DIS
LIN {X 43.203,Y -127.1356,Z 159,A -72.6178,B 21.2926,C -0.6917,E1 21.3565,E2 520.3078} C_DIS
LIN {X 46.3203,Y -126.0333,Z 159,A -71.3562,B 21.2927,C -0.6866,E1 21.3598,E2 519.0636} C_DIS
LIN {X 49.4262,Y -124.8479,Z 159,A -69.9407,B 21.2927,C -0.6883,E1 21.3634,E2 517.647} C_DIS
LIN {X 52.6846,Y -123.5071,Z 159,A -68.3529,B 21.2925,C -0.6944,E1 21.3676,E2 516.0468} C_DIS
LIN {X 55.8384,Y -122.1133,Z 159,A -66.9732,B 21.2925,C -0.6923,E1 21.371,E2 514.677} C_DIS
LIN {X 58.6438,Y -120.7926,Z 159,A -65.654,B 21.2925,C -0.6942,E1 21.3744,E2 513.3568} C_DIS
LIN {X 62.1119,Y -119.044,Z 159,A -63.9901,B 21.2925,C -0.6973,E1 21.3785,E2 511.69} C_DIS
LIN {X 65.922,Y -116.979,Z 159,A -62.1218,B 21.2923,C -0.7013,E1 21.3831,E2 509.8171} C_DIS
LIN {X 69.2336,Y -115.0503,Z 159,A -60.5293,B 21.2923,C -0.7022,E1 21.3869,E2 508.2279} C_DIS
LIN {X 72.3011,Y -113.1474,Z 159,A -58.9074,B 21.292,C -0.709,E1 21.3908,E2 506.5937} C_DIS
LIN {X 75.7392,Y -110.8757,Z 159,A -57.2441,B 21.292,C -0.7079,E1 21.3946,E2 504.9401} C_DIS
LIN {X 78.5627,Y -108.8933,Z 159,A -55.6681,B 21.2918,C -0.7158,E1 21.3982,E2 503.349} C_DIS
LIN {X 82.0269,Y -106.3083,Z 159,A -53.9425,B 21.2918,C -0.714,E1 21.402,E2 501.6358} C_DIS
LIN {X 85.1964,Y -103.7855,Z 159,A -52.1697,B 21.2917,C -0.7198,E1 21.4059,E2 499.855} C_DIS
LIN {X 88.5154,Y -100.9697,Z 159,A -50.3239,B 21.2916,C -0.7234,E1 21.4098,E2 498.0079} C_DIS
LIN {X 91.2928,Y -98.4656,Z 159,A -48.6771,B 21.2914,C -0.7296,E1 21.4132,E2 496.3524} C_DIS
LIN {X 94.4304,Y -95.4607,Z 159,A -46.8339,B 21.2912,C -0.7335,E1 21.4169,E2 494.5077} C_DIS
LIN {X 97.4694,Y -92.3556,Z 159,A -45.1016,B 21.2912,C -0.7321,E1 21.4202,E2 492.788} C_DIS
LIN {X 99.8265,Y -89.8027,Z 159,A -43.5114,B 21.291,C -0.741,E1 21.4232,E2 491.1819} C_DIS
LIN {X 102.746,Y -86.4469,Z 159,A -41.7529,B 21.291,C -0.7392,E1 21.4264,E2 489.438} C_DIS
LIN {X 105.2416,Y -83.391,Z 159,A -40.0539,B 21.2909,C -0.7443,E1 21.4294,E2 487.7344} C_DIS
LIN {X 107.5241,Y -80.4266,Z 159,A -38.3743,B 21.2906,C -0.7526,E1 21.4323,E2 486.0417} C_DIS
LIN {X 109.9745,Y -77.0426,Z 159,A -36.5835,B 21.2904,C -0.7578,E1 21.4352,E2 484.247} C_DIS
LIN {X 112.4638,Y -73.3604,Z 159,A -34.8314,B 21.2904,C -0.7561,E1 21.4378,E2 482.5101} C_DIS
LIN {X 114.303,Y -70.4604,Z 159,A -33.268,B 21.2902,C -0.7649,E1 21.4402,E2 480.9318} C_DIS
LIN {X 116.4212,Y -66.9033,Z 159,A -31.5394,B 21.2901,C -0.7681,E1 21.4426,E2 479.2052} C_DIS
LIN {X 118.4852,Y -63.1761,Z 159,A -29.7314,B 21.2899,C -0.7729,E1 21.445,E2 477.3954} C_DIS
LIN {X 120.1651,Y -59.9159,Z 159,A -28.2836,B 21.2899,C -0.7719,E1 21.4468,E2 475.9596} C_DIS
LIN {X 121.6844,Y -56.7659,Z 159,A -26.7691,B 21.2898,C -0.7774,E1 21.4486,E2 474.4398} C_DIS
LIN {X 123.0215,Y -53.8079,Z 159,A -25.414,B 21.2897,C -0.7801,E1 21.4502,E2 473.0862} C_DIS
LIN {X 124.3249,Y -50.7237,Z 159,A -23.9973,B 21.2895,C -0.7838,E1 21.4517,E2 471.6686} C_DIS
LIN {X 125.5451,Y -47.6235,Z 159,A -22.6886,B 21.2895,C -0.7827,E1 21.453,E2 470.3716} C_DIS
LIN {X 126.7381,Y -44.3495,Z 159,A -21.097,B 21.2892,C -0.7923,E1 21.4545,E2 468.7643} C_DIS
LIN {X 127.7364,Y -41.3884,Z 159,A -19.7923,B 21.2892,C -0.795,E1 21.4557,E2 467.461} C_DIS
LIN {X 128.7082,Y -38.2597,Z 159,A -18.4067,B 21.289,C -0.7988,E1 21.4568,E2 466.0745} C_DIS
LIN {X 129.637,Y -34.9816,Z 159,A -16.986,B 21.2889,C -0.8017,E1 21.4578,E2 464.6555} C_DIS
LIN {X 130.4836,Y -31.6763,Z 159,A -15.5389,B 21.2887,C -0.8059,E1 21.4588,E2 463.207} C_DIS
LIN {X 131.1909,Y -28.6068,Z 159,A -14.3875,B 21.2889,C -0.8008,E1 21.4595,E2 462.0775} C_DIS
LIN {X 131.7358,Y -25.993,Z 159,A -12.9778,B 21.2883,C -0.8175,E1 21.4603,E2 460.632} C_DIS
LIN {X 132.3127,Y -22.8758,Z 159,A -11.6398,B 21.2882,C -0.8211,E1 21.461,E2 459.2936} C_DIS
LIN {X 132.8243,Y -19.6861,Z 159,A -10.388,B 21.2882,C -0.8193,E1 21.4615,E2 458.0554} C_DIS
LIN {X 133.2659,Y -16.4265,Z 159,A -8.895,B 21.2879,C -0.8282,E1 21.462,E2 456.5488} C_DIS
LIN {X 133.7325,Y -12.0653,Z 159,A -7.022,B 21.2877,C -0.8342,E1 21.4625,E2 454.6725} C_DIS
LIN {X 134.008,Y -8.4416,Z 159,A -5.5796,B 21.2877,C -0.8339,E1 21.4628,E2 453.241} C_DIS
LIN {X 134.2076,Y -4.2377,Z 159,A -3.8896,B 21.2877,C -0.8345,E1 21.463,E2 451.5613} C_DIS
LIN {X 134.2723,Y -0.7533,Z 159,A -2.2294,B 21.2872,C -0.8477,E1 21.463,E2 449.8771} C_DIS
LIN {X 134.2287,Y 3.4802,Z 159,A -0.4778,B 21.2871,C -0.8508,E1 21.463,E2 448.1294} C_DIS
LIN {X 134.0662,Y 7.4977,Z 159,A 1.2564,B 21.2868,C -0.8571,E1 21.4628,E2 446.3902} C_DIS
LIN {X 133.834,Y 10.8642,Z 159,A 2.6579,B 21.2868,C -0.8598,E1 21.4625,E2 444.9912} C_DIS
LIN {X 133.5341,Y 14.0743,Z 159,A 4.0092,B 21.2866,C -0.863,E1 21.4621,E2 443.6408} C_DIS
LIN {X 133.1822,Y 17.0874,Z 159,A 5.2121,B 21.2866,C -0.8626,E1 21.4617,E2 442.4474} C_DIS
LIN {X 132.7786,Y 19.9878,Z 159,A 6.6079,B 21.2862,C -0.8736,E1 21.4611,E2 441.0314} C_DIS
LIN {X 132.2257,Y 23.3621,Z 159,A 7.9196,B 21.2862,C -0.8711,E1 21.4605,E2 439.7358} C_DIS
LIN {X 131.6844,Y 26.2454,Z 159,A 9.1998,B 21.2861,C -0.8763,E1 21.4598,E2 438.4502} C_DIS
LIN {X 131.0805,Y 29.118,Z 159,A 10.5291,B 21.2858,C -0.8839,E1 21.459,E2 437.1094} C_DIS
LIN {X 130.2473,Y 32.6359,Z 159,A 11.9834,B 21.2858,C -0.8843,E1 21.4581,E2 435.6639} C_DIS
LIN {X 129.3682,Y 35.9612,Z 159,A 13.2094,B 21.2861,C -0.8772,E1 21.4572,E2 434.4659} C_DIS
LIN {X 128.6341,Y 38.5128,Z 159,A 14.563,B 21.2855,C -0.8912,E1 21.4561,E2 433.0833} C_DIS
LIN {X 127.6306,Y 41.7165,Z 159,A 15.9571,B 21.2855,C -0.8936,E1 21.4549,E2 431.692} C_DIS
LIN {X 126.504,Y 45.0146,Z 159,A 17.5092,B 21.2851,C -0.9011,E1 21.4535,E2 430.1297} C_DIS
LIN {X 125.2471,Y 48.3994,Z 159,A 18.9697,B 21.2851,C -0.9018,E1 21.452,E2 428.677} C_DIS
LIN {X 124.0703,Y 51.342,Z 159,A 20.3313,B 21.2849,C -0.9062,E1 21.4506,E2 427.3126} C_DIS
LIN {X 122.8199,Y 54.2669,Z 159,A 21.7754,B 21.2846,C -0.9142,E1 21.449,E2 425.8559} C_DIS
LIN {X 121.4028,Y 57.3666,Z 159,A 23.0336,B 21.2848,C -0.9089,E1 21.4475,E2 424.6203} C_DIS
LIN {X 120.0441,Y 60.1612,Z 159,A 24.4547,B 21.2845,C -0.9171,E1 21.4458,E2 423.1857} C_DIS
LIN {X 118.1477,Y 63.8043,Z 159,A 26.2493,B 21.2842,C -0.9239,E1 21.4434,E2 421.3838} C_DIS
LIN {X 116.352,Y 67.0229,Z 159,A 27.7609,B 21.2842,C -0.9253,E1 21.4413,E2 419.878} C_DIS
LIN {X 114.303,Y 70.4604,Z 159,A 29.511,B 21.2838,C -0.9318,E1 21.4388,E2 418.1207} C_DIS
LIN {X 112.3117,Y 73.5931,Z 159,A 31.0335,B 21.2838,C -0.933,E1 21.4365,E2 416.604} C_DIS
LIN {X 110.3874,Y 76.4492,Z 159,A 32.6051,B 21.2834,C -0.9416,E1 21.434,E2 415.0181} C_DIS
LIN {X 107.8275,Y 80.019,Z 159,A 34.4546,B 21.2833,C -0.945,E1 21.4309,E2 413.1699} C_DIS
LIN {X 105.2416,Y 83.391,Z 159,A 36.2728,B 21.2831,C -0.9496,E1 21.4278,E2 411.3493} C_DIS
LIN {X 102.4553,Y 86.7913,Z 159,A 38.1253,B 21.283,C -0.9529,E1 21.4245,E2 409.498} C_DIS
LIN {X 99.6385,Y 90.0113,Z 159,A 39.8436,B 21.283,C -0.952,E1 21.4213,E2 407.7913} C_DIS
LIN {X 96.8697,Y 92.9844,Z 159,A 41.621,B 21.2827,C -0.9579,E1 21.4179,E2 406.0071} C_DIS
LIN {X 93.8106,Y 96.0699,Z 159,A 43.4655,B 21.2826,C -0.9614,E1 21.4143,E2 404.1623} C_DIS
LIN {X 90.7664,Y 98.9507,Z 159,A 45.2312,B 21.2825,C -0.964,E1 21.4106,E2 402.398} C_DIS
LIN {X 87.6046,Y 101.7605,Z 159,A 47.0473,B 21.2823,C -0.9681,E1 21.4068,E2 400.5793} C_DIS
LIN {X 84.5247,Y 104.3333,Z 159,A 48.6917,B 21.2823,C -0.9681,E1 21.4033,E2 398.9422} C_DIS
LIN {X 81.3401,Y 106.8346,Z 159,A 50.5039,B 21.282,C -0.9752,E1 21.3993,E2 397.1186} C_DIS
LIN {X 77.7475,Y 109.4773,Z 159,A 52.3054,B 21.282,C -0.9738,E1 21.3952,E2 395.3285} C_DIS
LIN {X 74.7416,Y 111.5505,Z 159,A 53.9345,B 21.2818,C -0.9797,E1 21.3914,E2 393.6899} C_DIS
LIN {X 71.2577,Y 113.8079,Z 159,A 55.7493,B 21.2816,C -0.9845,E1 21.3871,E2 391.869} C_DIS
LIN {X 67.368,Y 116.1522,Z 159,A 57.6367,B 21.2816,C -0.985,E1 21.3826,E2 389.987} C_DIS
LIN {X 63.6295,Y 118.2416,Z 159,A 59.535,B 21.2813,C -0.9908,E1 21.3779,E2 388.0793} C_DIS
LIN {X 59.9159,Y 120.1651,Z 159,A 61.0434,B 21.2818,C -0.9804,E1 21.3743,E2 386.6044} C_DIS
LIN {X 56.7468,Y 121.6932,Z 159,A 62.6125,B 21.2815,C -0.9854,E1 21.3703,E2 385.0266} C_DIS
LIN {X 53.8079,Y 123.0215,Z 159,A 64.013,B 21.2815,C -0.9881,E1 21.3667,E2 383.6228} C_DIS
LIN {X 50.7237,Y 124.3249,Z 159,A 65.4364,B 21.2814,C -0.9894,E1 21.363,E2 382.1998} C_DIS
LIN {X 47.3604,Y 125.6437,Z 159,A 66.9305,B 21.2814,C -0.9888,E1 21.3592,E2 380.7113} C_DIS
LIN {X 44.3574,Y 126.7353,Z 159,A 68.2806,B 21.2814,C -0.9894,E1 21.3556,E2 379.3628} C_DIS
LIN {X 41.3884,Y 127.7364,Z 159,A 69.6634,B 21.2812,C -0.9926,E1 21.3519,E2 377.9743} C_DIS
LIN {X 38.2597,Y 128.7082,Z 159,A 71.057,B 21.2812,C -0.9935,E1 21.3482,E2 376.5813} C_DIS
LIN {X 34.9173,Y 129.6541,Z 159,A 72.5441,B 21.2812,C -0.9948,E1 21.3442,E2 375.0936} C_DIS
LIN {X 32.0837,Y 130.3854,Z 159,A 73.809,B 21.2811,C -0.9962,E1 21.3408,E2 373.8268} C_DIS
LIN {X 29.118,Y 131.0805,Z 159,A 75.0763,B 21.2811,C -0.9955,E1 21.3373,E2 372.5637} C_DIS
LIN {X 25.7475,Y 131.7827,Z 159,A 76.6336,B 21.2809,C -1.0002,E1 21.333,E2 370.9958} C_DIS
LIN {X 22.3114,Y 132.4069,Z 159,A 77.9958,B 21.2811,C -0.995,E1 21.3293,E2 369.6496} C_DIS
LIN {X 19.4378,Y 132.8598,Z 159,A 79.2857,B 21.2811,C -0.9976,E1 21.3258,E2 368.3541} C_DIS
LIN {X 16.4265,Y 133.2659,Z 159,A 80.6455,B 21.2809,C -1.0007,E1 21.322,E2 366.9868} C_DIS
LIN {X 12.95,Y 133.6476,Z 159,A 82.0686,B 21.2809,C -0.9979,E1 21.318,E2 365.5727} C_DIS
LIN {X 8.7697,Y 133.9878,Z 159,A 83.741,B 21.2812,C -0.9928,E1 21.3134,E2 363.9153} C_DIS
LIN {X 5.986,Y 134.1422,Z 159,A 85.188,B 21.2807,C -1.0042,E1 21.3093,E2 362.4375} C_DIS
LIN {X 2.1022,Y 134.2572,Z 159,A 86.7443,B 21.2809,C -0.9996,E1 21.305,E2 360.8942} C_DIS
LIN {X -1.4869,Y 134.2674,Z 159,A 88.2097,B 21.2811,C -0.9964,E1 21.3009,E2 359.4377} C_DIS
LIN {X -4.7236,Y 134.1914,Z 159,A 89.6106,B 21.2811,C -0.9969,E1 21.297,E2 358.0352} C_DIS
LIN {X -7.9579,Y 134.0378,Z 159,A 91.0179,B 21.2811,C -0.9976,E1 21.2931,E2 356.6256} C_DIS
LIN {X -10.9997,Y 133.8225,Z 159,A 92.3027,B 21.2811,C -0.9963,E1 21.2895,E2 355.3435} C_DIS
LIN {X -15.6737,Y 133.3557,Z 159,A 94.2713,B 21.2811,C -0.9938,E1 21.2841,E2 353.3806} C_DIS
LIN {X -18.5376,Y 132.9884,Z 159,A 95.5996,B 21.2811,C -0.9973,E1 21.2804,E2 352.0415} C_DIS
LIN {X -22.0235,Y 132.4549,Z 159,A 96.9069,B 21.2814,C -0.9876,E1 21.2768,E2 350.7593} C_DIS
LIN {X -24.6854,Y 131.9858,Z 159,A 98.2756,B 21.2811,C -0.9962,E1 21.273,E2 349.3654} C_DIS
LIN {X -27.8074,Y 131.3634,Z 159,A 99.4632,B 21.2814,C -0.9877,E1 21.2698,E2 348.1996} C_DIS
LIN {X -30.9358,Y 130.6621,Z 159,A 100.9713,B 21.2812,C -0.9926,E1 21.2657,E2 346.6757} C_DIS
LIN {X -34.3674,Y 129.8008,Z 159,A 102.2322,B 21.2818,C -0.9803,E1 21.2623,E2 345.4462} C_DIS
LIN {X -36.9471,Y 129.0925,Z 159,A 103.5969,B 21.2814,C -0.9888,E1 21.2586,E2 344.0556} C_DIS
LIN {X -40.0776,Y 128.1551,Z 159,A 104.9971,B 21.2814,C -0.9876,E1 21.2549,E2 342.656} C_DIS
LIN {X -43.203,Y 127.1356,Z 159,A 106.4936,B 21.2814,C -0.99,E1 21.2509,E2 341.1495} C_DIS
LIN {X -46.6414,Y 125.913,Z 159,A 108.03,B 21.2814,C -0.9872,E1 21.2468,E2 339.6172} C_DIS
LIN {X -49.4262,Y 124.8479,Z 159,A 109.2473,B 21.2816,C -0.9831,E1 21.2437,E2 338.408} C_DIS
LIN {X -52.5175,Y 123.5794,Z 159,A 110.8122,B 21.2815,C -0.9871,E1 21.2396,E2 336.8277} C_DIS
LIN {X -56.0512,Y 122.0148,Z 159,A 112.3501,B 21.2818,C -0.98,E1 21.2358,E2 335.305} C_DIS
LIN {X -59.146,Y 120.5449,Z 159,A 113.7295,B 21.282,C -0.9742,E1 21.2323,E2 333.9374} C_DIS
LIN {X -61.6721,Y 119.2749,Z 159,A 115.1613,B 21.2817,C -0.9819,E1 21.2287,E2 332.4797} C_DIS
LIN {X -65.5385,Y 117.1945,Z 159,A 117.0177,B 21.2819,C -0.978,E1 21.2242,E2 330.6276} C_DIS
LIN {X -69.2336,Y 115.0503,Z 159,A 118.7325,B 21.2822,C -0.9702,E1 21.2201,E2 328.9282} C_DIS
LIN {X -72.1496,Y 113.2444,Z 159,A 120.2037,B 21.2823,C -0.9679,E1 21.2166,E2 327.458} C_DIS
LIN {X -75.515,Y 111.0286,Z 159,A 122.0247,B 21.2823,C -0.9689,E1 21.2124,E2 325.6269} C_DIS
LIN {X -79.149,Y 108.4684,Z 159,A 123.9359,B 21.2824,C -0.9657,E1 21.208,E2 323.7165} C_DIS
LIN {X -82.6004,Y 105.8637,Z 159,A 125.6944,B 21.2827,C -0.9582,E1 21.2042,E2 321.9711} C_DIS
LIN {X -85.4129,Y 103.6074,Z 159,A 127.3496,B 21.2827,C -0.9599,E1 21.2005,E2 320.3039} C_DIS
LIN {X -88.7151,Y 100.7943,Z 159,A 129.1032,B 21.283,C -0.9517,E1 21.1969,E2 318.5647} C_DIS
LIN {X -91.2928,Y 98.4656,Z 159,A 130.7063,B 21.283,C -0.9534,E1 21.1935,E2 316.9491} C_DIS
LIN {X -94.4304,Y 95.4607,Z 159,A 132.579,B 21.283,C -0.9499,E1 21.1898,E2 315.0769} C_DIS
LIN {X -97.4694,Y 92.3556,Z 159,A 134.3236,B 21.2835,C -0.9408,E1 21.1865,E2 313.3483} C_DIS
LIN {X -99.8265,Y 89.8027,Z 159,A 135.815,B 21.2836,C -0.9375,E1 21.1837,E2 311.8582} C_DIS
LIN {X -102.4954,Y 86.7442,Z 159,A 137.6113,B 21.2836,C -0.9358,E1 21.1804,E2 310.0568} C_DIS
LIN {X -105.2416,Y 83.391,Z 159,A 139.4347,B 21.2839,C -0.93,E1 21.1772,E2 308.2394} C_DIS
LIN {X -107.5241,Y 80.4266,Z 159,A 141.1366,B 21.2839,C -0.9301,E1 21.1743,E2 306.5273} C_DIS
LIN {X -109.9745,Y 77.0426,Z 159,A 142.927,B 21.2841,C -0.9257,E1 21.1714,E2 304.7389} C_DIS
LIN {X -112.3881,Y 73.477,Z 159,A 144.7525,B 21.2843,C -0.9201,E1 21.1686,E2 302.9178} C_DIS
LIN {X -114.6788,Y 69.848,Z 159,A 146.5675,B 21.2846,C -0.9143,E1 21.1659,E2 301.1078} C_DIS
LIN {X -116.8442,Y 66.1619,Z 159,A 148.3823,B 21.2848,C -0.9087,E1 21.1634,E2 299.2971} C_DIS
LIN {X -118.6128,Y 62.933,Z 159,A 149.9263,B 21.285,C -0.9031,E1 21.1614,E2 297.759} C_DIS
LIN {X -120.1651,Y 59.9159,Z 159,A 151.2789,B 21.2854,C -0.8949,E1 21.1597,E2 296.4203} C_DIS
LIN {X -121.5205,Y 57.1203,Z 159,A 152.8666,B 21.2851,C -0.9019,E1 21.1577,E2 294.8031} C_DIS
LIN {X -123.0661,Y 53.7046,Z 159,A 154.2918,B 21.2856,C -0.8899,E1 21.1561,E2 293.4017} C_DIS
LIN {X -124.3249,Y 50.7237,Z 159,A 155.7169,B 21.2856,C -0.8876,E1 21.1546,E2 291.9736} C_DIS
LIN {X -125.5451,Y 47.6235,Z 159,A 157.2201,B 21.2856,C -0.8866,E1 21.1531,E2 290.4628} C_DIS
LIN {X -126.7864,Y 44.2101,Z 159,A 158.6097,B 21.2861,C -0.8753,E1 21.1518,E2 289.0953} C_DIS
LIN {X -127.7364,Y 41.3884,Z 159,A 159.9855,B 21.2861,C -0.8757,E1 21.1506,E2 287.709} C_DIS
LIN {X -128.7082,Y 38.2597,Z 159,A 161.3924,B 21.2863,C -0.8717,E1 21.1495,E2 286.3033} C_DIS
LIN {X -129.5305,Y 35.3808,Z 159,A 162.8313,B 21.2862,C -0.8744,E1 21.1484,E2 284.847} C_DIS
LIN {X -130.3457,Y 32.2483,Z 159,A 164.1538,B 21.2864,C -0.8676,E1 21.1475,E2 283.534} C_DIS
LIN {X -131.0805,Y 29.118,Z 159,A 165.4491,B 21.2867,C -0.8602,E1 21.1467,E2 282.2504} C_DIS
LIN {X -131.8087,Y 25.6115,Z 159,A 166.838,B 21.2871,C -0.8496,E1 21.1459,E2 280.8809} C_DIS
LIN {X -132.3127,Y 22.8758,Z 159,A 168.2648,B 21.2869,C -0.8557,E1 21.1452,E2 279.4271} C_DIS
LIN {X -132.89,Y 19.2265,Z 159,A 169.7816,B 21.2872,C -0.8483,E1 21.1446,E2 277.92} C_DIS
LIN {X -133.2659,Y 16.4265,Z 159,A 170.9796,B 21.2873,C -0.8441,E1 21.1442,E2 276.7251} C_DIS
LIN {X -133.6092,Y 13.3499,Z 159,A 172.2137,B 21.2876,C -0.8363,E1 21.1438,E2 275.5037} C_DIS
LIN {X -133.8615,Y 10.5376,Z 159,A 173.6475,B 21.2874,C -0.8419,E1 21.1435,E2 274.0441} C_DIS
LIN {X -134.0967,Y 6.8904,Z 159,A 175.1262,B 21.2877,C -0.8336,E1 21.1432,E2 272.5777} C_DIS
LIN {X -134.2299,Y 3.4362,Z 159,A 176.6139,B 21.2879,C -0.8294,E1 21.1432,E2 271.0909} C_DIS
LIN {X -134.2759,Y 0,Z 159,A 178.0571,B 21.2881,C -0.8238,E1 21.1431,E2 269.653} C_DIS
LIN {X -134.2426,Y -2.9804,Z 159,A 179.4188,B 21.2881,C -0.8234,E1 21.1431,E2 268.2824} C_DIS
LIN {X -134.1143,Y -6.5409,Z 159,A -179.086,B 21.2883,C -0.8176,E1 21.1433,E2 266.7927} C_DIS
LIN {X -133.9249,Y -9.6703,Z 159,A -177.9018,B 21.2887,C -0.807,E1 21.1435,E2 265.6292} C_DIS
LIN {X -133.7325,Y -12.0653,Z 159,A -176.6348,B 21.2885,C -0.8137,E1 21.1439,E2 264.3345} C_DIS
LIN {X -133.42,Y -15.1345,Z 159,A -175.3319,B 21.2886,C -0.809,E1 21.1443,E2 263.0353} C_DIS
LIN {X -132.9979,Y -18.4709,Z 159,A -173.8686,B 21.2888,C -0.8057,E1 21.1448,E2 261.5707} C_DIS
LIN {X -132.464,Y -21.9692,Z 159,A -172.5629,B 21.2892,C -0.7926,E1 21.1454,E2 260.2922} C_DIS
LIN {X -131.9858,Y -24.6854,Z 159,A -171.2541,B 21.2892,C -0.7944,E1 21.146,E2 258.9692} C_DIS
LIN {X -131.3634,Y -27.8074,Z 159,A -169.9828,B 21.2894,C -0.7866,E1 21.1467,E2 257.7105} C_DIS
LIN {X -130.6621,Y -30.9358,Z 159,A -168.6028,B 21.2896,C -0.7829,E1 21.1476,E2 256.331} C_DIS
LIN {X -129.8288,Y -34.2623,Z 159,A -167.2041,B 21.2898,C -0.7757,E1 21.1485,E2 254.9424} C_DIS
LIN {X -129.0925,Y -36.9471,Z 159,A -165.8277,B 21.2897,C -0.7799,E1 21.1496,E2 253.5448} C_DIS
LIN {X -128.154,Y -40.0812,Z 159,A -164.2806,B 21.2896,C -0.7821,E1 21.1509,E2 251.9811} C_DIS
LIN {X -126.961,Y -43.7066,Z 159,A -162.7602,B 21.2899,C -0.7728,E1 21.1522,E2 250.4761} C_DIS
LIN {X -126.0333,Y -46.3203,Z 159,A -161.5832,B 21.29,C -0.769,E1 21.1533,E2 249.3016} C_DIS
LIN {X -124.652,Y -49.9121,Z 159,A -159.9647,B 21.2902,C -0.7633,E1 21.155,E2 247.6881} C_DIS
LIN {X -123.3509,Y -53.0459,Z 159,A -158.6884,B 21.2906,C -0.752,E1 21.1563,E2 246.4347} C_DIS
LIN {X -122.1133,Y -55.8384,Z 159,A -157.1538,B 21.2904,C -0.7579,E1 21.1581,E2 244.8735} C_DIS
LIN {X -120.7926,Y -58.6438,Z 159,A -155.8204,B 21.2905,C -0.7546,E1 21.1597,E2 243.5406} C_DIS
LIN {X -119.1001,Y -62.005,Z 159,A -154.1554,B 21.2906,C -0.7527,E1 21.1618,E2 241.8701} C_DIS
LIN {X -116.9425,Y -65.9869,Z 159,A -152.2073,B 21.2908,C -0.7481,E1 21.1645,E2 239.9225} C_DIS
LIN {X -114.892,Y -69.4953,Z 159,A -150.4461,B 21.2908,C -0.7447,E1 21.167,E2 238.1599} C_DIS
LIN {X -112.5295,Y -73.2593,Z 159,A -148.5276,B 21.291,C -0.7407,E1 21.1699,E2 236.2408} C_DIS
LIN {X -110.3874,Y -76.4492,Z 159,A -146.8299,B 21.291,C -0.7391,E1 21.1726,E2 234.5377} C_DIS
LIN {X -107.7895,Y -80.07,Z 159,A -144.9359,B 21.2912,C -0.7341,E1 21.1757,E2 232.6465} C_DIS
LIN {X -105.1131,Y -83.5524,Z 159,A -143.064,B 21.2914,C -0.7295,E1 21.1789,E2 230.7767} C_DIS
LIN {X -102.4954,Y -86.7442,Z 159,A -141.264,B 21.2914,C -0.727,E1 21.1821,E2 228.9736} C_DIS
LIN {X -99.6385,Y -90.0113,Z 159,A -139.4058,B 21.2916,C -0.7231,E1 21.1856,E2 227.1163} C_DIS
LIN {X -96.5808,Y -93.2842,Z 159,A -137.4919,B 21.2917,C -0.7191,E1 21.1893,E2 225.2036} C_DIS
LIN {X -93.4247,Y -96.4448,Z 159,A -135.6021,B 21.2919,C -0.7144,E1 21.193,E2 223.3173} C_DIS
LIN {X -90.2938,Y -99.3821,Z 159,A -133.7508,B 21.2919,C -0.7115,E1 21.1968,E2 221.465} C_DIS
LIN {X -87.2983,Y -102.0243,Z 159,A -132.1054,B 21.2921,C -0.7057,E1 21.2003,E2 219.8281} C_DIS
LIN {X -84.5247,Y -104.3333,Z 159,A -130.576,B 21.2922,C -0.7023,E1 21.2036,E2 218.3011} C_DIS
LIN {X -81.2836,Y -106.8779,Z 159,A -128.7211,B 21.2922,C -0.7033,E1 21.2077,E2 216.4352} C_DIS
LIN {X -77.7475,Y -109.4773,Z 159,A -126.8523,B 21.2923,C -0.7,E1 21.2119,E2 214.5679} C_DIS
LIN {X -74.1953,Y -111.9152,Z 159,A -124.9965,B 21.2923,C -0.6977,E1 21.2162,E2 212.7109} C_DIS
LIN {X -70.5785,Y -114.2306,Z 159,A -123.2478,B 21.2926,C -0.6913,E1 21.2203,E2 210.9734} C_DIS
LIN {X -67.4395,Y -116.1108,Z 159,A -121.576,B 21.2926,C -0.6939,E1 21.2244,E2 209.2885} C_DIS
LIN {X -63.8043,Y -118.1477,Z 159,A -119.7715,B 21.2926,C -0.6926,E1 21.2288,E2 207.4813} C_DIS
LIN {X -59.719,Y -120.2623,Z 159,A -117.9731,B 21.2928,C -0.6829,E1 21.2332,E2 205.7039} C_DIS
LIN {X -57.1203,Y -121.5205,Z 159,A -116.6084,B 21.2928,C -0.6872,E1 21.2367,E2 204.3231} C_DIS
LIN {X -53.8079,Y -123.0215,Z 159,A -115.1432,B 21.2928,C -0.6817,E1 21.2404,E2 202.8688} C_DIS
LIN {X -50.5325,Y -124.402,Z 159,A -113.6006,B 21.2928,C -0.6813,E1 21.2444,E2 201.3233} C_DIS
LIN {X -47.4564,Y -125.6077,Z 159,A -112.3824,B 21.2932,C -0.6715,E1 21.2475,E2 200.1291} C_DIS
LIN {X -44.5107,Y -126.6822,Z 159,A -110.8736,B 21.293,C -0.6778,E1 21.2515,E2 198.5992} C_DIS
LIN {X -41.3884,Y -127.7364,Z 159,A -109.4665,B 21.293,C -0.6767,E1 21.2553,E2 197.1921} C_DIS
LIN {X -38.0379,Y -128.7731,Z 159,A -107.9747,B 21.293,C -0.6754,E1 21.2592,E2 195.7008} C_DIS
LIN {X -35.2062,Y -129.5771,Z 159,A -106.6866,B 21.293,C -0.676,E1 21.2627,E2 194.4086} C_DIS
LIN {X -32.2483,Y -130.3457,Z 159,A -105.3235,B 21.293,C -0.6779,E1 21.2664,E2 193.0381} C_DIS
LIN {X -28.7262,Y -131.1651,Z 159,A -103.8774,B 21.2932,C -0.6728,E1 21.2703,E2 191.6039} C_DIS
LIN {X -25.6951,Y -131.7927,Z 159,A -102.5624,B 21.2932,C -0.672,E1 21.2739,E2 190.2894} C_DIS
LIN {X -22.8758,Y -132.3127,Z 159,A -101.2401,B 21.2931,C -0.6759,E1 21.2776,E2 188.9545} C_DIS
LIN {X -19.5252,Y -132.8473,Z 159,A -99.8173,B 21.2931,C -0.6744,E1 21.2815,E2 187.5344} C_DIS
LIN {X -15.9918,Y -133.3177,Z 159,A -98.3759,B 21.2932,C -0.6706,E1 21.2855,E2 186.1025} C_DIS
LIN {X -13.3499,Y -133.6092,Z 159,A -97.3196,B 21.2933,C -0.6669,E1 21.2884,E2 185.0556} C_DIS
LIN {X -10.5376,Y -133.8615,Z 159,A -95.9422,B 21.2931,C -0.6746,E1 21.2923,E2 183.6562} C_DIS
LIN {X -7.4977,Y -134.0662,Z 159,A -94.605,B 21.2931,C -0.6763,E1 21.296,E2 182.3138} C_DIS
LIN {X -3.9559,Y -134.2155,Z 159,A -93.2013,B 21.2931,C -0.6715,E1 21.2999,E2 180.9231} C_DIS
LIN {X 0.9317,Y -134.2705,Z 159,A -91.486,B 21.2937,C -0.6551,E1 21.3046,E2 179.2529} C_DIS
Enddeposition()
LIN {X 0.9317,Y -134.2705,Z 159,A -91.486,B 21.2937,C -0.6551,E1 21.3046,E2 179.2529} C_DIS
Startdeposition()
$VEL.CP = VEL_PRINT
LIN {X 0.4977,Y -133.3449,Z 159,A -91.7032,B 20.1882,C -0.4938,E1 20.1937,E2 179.8182} C_DIS
LIN {X -3.7107,Y -133.294,Z 159,A -93.4269,B 20.1881,C -0.4971,E1 20.1889,E2 181.5325} C_DIS
LIN {X -7.9521,Y -133.1085,Z 159,A -95.1654,B 20.1881,C -0.5006,E1 20.184,E2 183.2612} C_DIS
LIN {X -11.3572,Y -132.8611,Z 159,A -96.7773,B 20.1881,C -0.4947,E1 20.1795,E2 184.8914} C_DIS
LIN {X -15.6876,Y -132.4195,Z 159,A -98.5694,B 20.1881,C -0.4982,E1 20.1746,E2 186.6745} C_DIS
LIN {X -19.1891,Y -131.9579,Z 159,A -100.1874,B 20.1881,C -0.4944,E1 20.17,E2 188.3052} C_DIS
LIN {X -23.1223,Y -131.3259,Z 159,A -101.8379,B 20.1881,C -0.4975,E1 20.1655,E2 189.9487} C_DIS
LIN {X -26.7059,Y -130.6437,Z 159,A -103.3526,B 20.1881,C -0.5004,E1 20.1614,E2 191.4572} C_DIS
LIN {X -29.7912,Y -129.9749,Z 159,A -104.76,B 20.1881,C -0.4989,E1 20.1575,E2 192.871} C_DIS
LIN {X -34.9509,Y -128.6848,Z 159,A -107.1038,B 20.1881,C -0.4979,E1 20.1512,E2 195.2222} C_DIS
LIN {X -38.4913,Y -127.6702,Z 159,A -108.6777,B 20.1881,C -0.4993,E1 20.147,E2 196.7951} C_DIS
LIN {X -42.9965,Y -126.225,Z 159,A -110.6811,B 20.188,C -0.5022,E1 20.1417,E2 198.795} C_DIS
LIN {X -46.6459,Y -124.9204,Z 159,A -112.2955,B 20.1879,C -0.5058,E1 20.1374,E2 200.403} C_DIS
LIN {X -49.6603,Y -123.7531,Z 159,A -113.6867,B 20.1879,C -0.507,E1 20.1338,E2 201.7943} C_DIS
LIN {X -52.7636,Y -122.462,Z 159,A -115.0531,B 20.1877,C -0.5117,E1 20.1303,E2 203.151} C_DIS
LIN {X -55.4513,Y -121.2699,Z 159,A -116.485,B 20.1879,C -0.5063,E1 20.1266,E2 204.6032} C_DIS
LIN {X -58.7628,Y -119.6992,Z 159,A -117.9711,B 20.1877,C -0.5118,E1 20.1229,E2 206.0781} C_DIS
LIN {X -61.4553,Y -118.3407,Z 159,A -119.3594,B 20.1877,C -0.5097,E1 20.1195,E2 207.4774} C_DIS
LIN {X -65.3366,Y -116.2435,Z 159,A -121.1851,B 20.1877,C -0.5151,E1 20.115,E2 209.294} C_DIS
LIN {X -68.4421,Y -114.4428,Z 159,A -122.8069,B 20.1877,C -0.5141,E1 20.1111,E2 210.9249} C_DIS
LIN {X -72.0105,Y -112.2316,Z 159,A -124.6344,B 20.1877,C -0.5159,E1 20.1068,E2 212.7545} C_DIS
LIN {X -75.7673,Y -109.731,Z 159,A -126.6269,B 20.1877,C -0.5168,E1 20.1021,E2 214.7526} C_DIS
LIN {X -79.3926,Y -107.137,Z 159,A -128.5289,B 20.1875,C -0.5207,E1 20.0979,E2 216.652} C_DIS
LIN {X -82.6543,Y -104.6414,Z 159,A -130.2514,B 20.1875,C -0.5255,E1 20.0941,E2 218.3684} C_DIS
LIN {X -86.4418,Y -101.5344,Z 159,A -132.3401,B 20.1873,C -0.5301,E1 20.0896,E2 220.4538} C_DIS
LIN {X -89.4624,Y -98.8835,Z 159,A -134.1183,B 20.1873,C -0.5314,E1 20.0859,E2 222.237} C_DIS
LIN {X -93.0104,Y -95.5542,Z 159,A -136.2622,B 20.1873,C -0.5336,E1 20.0815,E2 224.3859} C_DIS
LIN {X -96.1053,Y -92.4413,Z 159,A -138.1711,B 20.1871,C -0.5367,E1 20.0778,E2 226.2962} C_DIS
LIN {X -99.1408,Y -89.1773,Z 159,A -139.7558,B 20.1867,C -0.5539,E1 20.0749,E2 227.8394} C_DIS
LIN {X -101.3925,Y -86.6088,Z 159,A -141.5767,B 20.187,C -0.5433,E1 20.0715,E2 229.7017} C_DIS
LIN {X -103.8743,Y -83.6156,Z 159,A -143.1274,B 20.1867,C -0.5519,E1 20.0688,E2 231.2364} C_DIS
LIN {X -106.3963,Y -80.382,Z 159,A -144.9764,B 20.1867,C -0.5527,E1 20.0656,E2 233.0943} C_DIS
LIN {X -108.8625,Y -77.0091,Z 159,A -146.7825,B 20.1867,C -0.5567,E1 20.0626,E2 234.8999} C_DIS
LIN {X -110.4158,Y -74.7648,Z 159,A -148.0941,B 20.1867,C -0.5542,E1 20.0606,E2 236.227} C_DIS
LIN {X -112.9581,Y -70.8663,Z 159,A -150.0292,B 20.1865,C -0.5619,E1 20.0577,E2 238.1523} C_DIS
LIN {X -115.05,Y -67.4163,Z 159,A -151.679,B 20.1863,C -0.5697,E1 20.0553,E2 239.7901} C_DIS
LIN {X -117.1491,Y -63.699,Z 159,A -153.5917,B 20.1863,C -0.5715,E1 20.0527,E2 241.7102} C_DIS
LIN {X -118.6778,Y -60.7996,Z 159,A -154.8997,B 20.186,C -0.5793,E1 20.0511,E2 243.0045} C_DIS
LIN {X -119.7935,Y -58.5716,Z 159,A -156.2824,B 20.1862,C -0.5701,E1 20.0493,E2 244.4233} C_DIS
LIN {X -121.9814,Y -53.8689,Z 159,A -158.3445,B 20.1859,C -0.5828,E1 20.047,E2 246.4629} C_DIS
LIN {X -123.5835,Y -50.0809,Z 159,A -159.9172,B 20.1856,C -0.5953,E1 20.0453,E2 248.0101} C_DIS
LIN {X -124.4261,Y -47.9502,Z 159,A -161.0832,B 20.1856,C -0.5911,E1 20.0441,E2 249.1965} C_DIS
LIN {X -125.9022,Y -43.9276,Z 159,A -162.8747,B 20.1855,C -0.5984,E1 20.0424,E2 250.9797} C_DIS
LIN {X -126.9886,Y -40.6798,Z 159,A -164.283,B 20.1853,C -0.6052,E1 20.0412,E2 252.3784} C_DIS
LIN {X -127.7967,Y -38.0702,Z 159,A -165.4452,B 20.1852,C -0.6091,E1 20.0403,E2 253.5377} C_DIS
LIN {X -128.762,Y -34.6611,Z 159,A -167.1006,B 20.1852,C -0.6085,E1 20.039,E2 255.2069} C_DIS
LIN {X -129.6388,Y -31.2211,Z 159,A -168.4938,B 20.1849,C -0.6182,E1 20.0381,E2 256.5822} C_DIS
LIN {X -130.974,Y -25.036,Z 159,A -171.3995,B 20.1849,C -0.6193,E1 20.0364,E2 259.5064} C_DIS
LIN {X -131.7235,Y -20.7369,Z 159,A -173.2492,B 20.1847,C -0.6261,E1 20.0356,E2 261.3504} C_DIS
LIN {X -132.5708,Y -14.3532,Z 159,A -176.0221,B 20.1844,C -0.6344,E1 20.0346,E2 264.12} C_DIS
LIN {X -133.0463,Y -8.9594,Z 159,A -178.4825,B 20.1844,C -0.6366,E1 20.034,E2 266.5929} C_DIS
LIN {X -133.2409,Y -5.2838,Z 159,A 179.926,B 20.1842,C -0.6412,E1 20.0338,E2 268.1831} C_DIS
LIN {X -133.3452,Y -0.5659,Z 159,A 178.0213,B 20.1839,C -0.6523,E1 20.0338,E2 270.07} C_DIS
LIN {X -133.3059,Y 3.2812,Z 159,A 176.2702,B 20.1839,C -0.6537,E1 20.0338,E2 271.8302} C_DIS
LIN {X -133.1591,Y 7.0584,Z 159,A 174.5547,B 20.1838,C -0.6554,E1 20.0341,E2 273.554} C_DIS
LIN {X -132.8505,Y 11.4817,Z 159,A 172.6466,B 20.1836,C -0.6613,E1 20.0345,E2 275.4594} C_DIS
LIN {X -132.4688,Y 15.2742,Z 159,A 170.8366,B 20.1836,C -0.6599,E1 20.035,E2 277.2872} C_DIS
LIN {X -131.8573,Y 19.8729,Z 159,A 169.2254,B 20.183,C -0.6807,E1 20.0356,E2 278.8499} C_DIS
LIN {X -131.1709,Y 23.9843,Z 159,A 167.2726,B 20.183,C -0.6802,E1 20.0366,E2 280.819} C_DIS
LIN {X -130.6973,Y 26.4425,Z 159,A 165.5215,B 20.1837,C -0.658,E1 20.0376,E2 282.648} C_DIS
LIN {X -129.5435,Y 31.6163,Z 159,A 163.823,B 20.1828,C -0.6869,E1 20.0387,E2 284.2747} C_DIS
LIN {X -128.5099,Y 35.5846,Z 159,A 162.334,B 20.1822,C -0.7028,E1 20.0397,E2 285.7284} C_DIS
LIN {X -127.5802,Y 38.7855,Z 159,A 160.6835,B 20.1824,C -0.6988,E1 20.041,E2 287.4025} C_DIS
LIN {X -126.6556,Y 41.7071,Z 159,A 159.3411,B 20.1823,C -0.7018,E1 20.0422,E2 288.7458} C_DIS
LIN {X -125.4961,Y 45.0742,Z 159,A 158.0613,B 20.1818,C -0.7161,E1 20.0433,E2 289.9933} C_DIS
LIN {X -124.3537,Y 48.1364,Z 159,A 156.3919,B 20.182,C -0.7101,E1 20.045,E2 291.692} C_DIS
LIN {X -123.2851,Y 50.8143,Z 159,A 154.8438,B 20.1823,C -0.702,E1 20.0467,E2 293.2748} C_DIS
LIN {X -121.9687,Y 53.8971,Z 159,A 153.6884,B 20.1818,C -0.7171,E1 20.0479,E2 294.3942} C_DIS
LIN {X -120.8439,Y 56.3724,Z 159,A 152.1795,B 20.1821,C -0.7076,E1 20.0498,E2 295.9413} C_DIS
LIN {X -119.2633,Y 59.6465,Z 159,A 150.8067,B 20.1817,C -0.7193,E1 20.0514,E2 297.2894} C_DIS
LIN {X -116.5039,Y 64.872,Z 159,A 148.3071,B 20.1814,C -0.728,E1 20.0547,E2 299.7803} C_DIS
LIN {X -114.2798,Y 68.7144,Z 159,A 146.3489,B 20.1813,C -0.7314,E1 20.0575,E2 301.7414} C_DIS
LIN {X -111.8083,Y 72.6659,Z 159,A 144.3753,B 20.181,C -0.738,E1 20.0605,E2 303.7084} C_DIS
LIN {X -109.2408,Y 76.4724,Z 159,A 142.3464,B 20.181,C -0.7412,E1 20.0637,E2 305.7409} C_DIS
LIN {X -106.6437,Y 80.0542,Z 159,A 140.4399,B 20.1808,C -0.7459,E1 20.0668,E2 307.6452} C_DIS
LIN {X -103.8988,Y 83.5852,Z 159,A 138.5542,B 20.1805,C -0.7523,E1 20.0701,E2 309.5237} C_DIS
LIN {X -101.2967,Y 86.7212,Z 159,A 136.7787,B 20.1805,C -0.7557,E1 20.0733,E2 311.2994} C_DIS
LIN {X -98.5412,Y 89.8397,Z 159,A 134.9318,B 20.1803,C -0.7578,E1 20.0767,E2 313.1506} C_DIS
LIN {X -95.4183,Y 93.1497,Z 159,A 132.9289,B 20.1803,C -0.7606,E1 20.0806,E2 315.1563} C_DIS
LIN {X -90.7348,Y 97.7173,Z 159,A 129.8044,B 20.1804,C -0.755,E1 20.087,E2 318.3137} C_DIS
LIN {X -87.6757,Y 100.4709,Z 159,A 128.4065,B 20.1798,C -0.7732,E1 20.0898,E2 319.6655} C_DIS
LIN {X -84.2375,Y 103.3707,Z 159,A 126.4484,B 20.1797,C -0.7763,E1 20.094,E2 321.624} C_DIS
LIN {X -81.0653,Y 105.8765,Z 159,A 124.7177,B 20.1795,C -0.7801,E1 20.0979,E2 323.3516} C_DIS
LIN {X -77.3976,Y 108.5867,Z 159,A 122.7788,B 20.1793,C -0.7848,E1 20.1022,E2 325.2855} C_DIS
LIN {X -73.8656,Y 111.0196,Z 159,A 120.9284,B 20.1793,C -0.788,E1 20.1065,E2 327.1344} C_DIS
LIN {X -70.1583,Y 113.3991,Z 159,A 119.0028,B 20.1791,C -0.7901,E1 20.111,E2 329.0616} C_DIS
LIN {X -66.5496,Y 115.5537,Z 159,A 117.1698,B 20.1791,C -0.7922,E1 20.1155,E2 330.8956} C_DIS
LIN {X -63.2356,Y 117.3998,Z 159,A 115.6635,B 20.1788,C -0.7997,E1 20.1191,E2 332.3853} C_DIS
LIN {X -59.2079,Y 119.4796,Z 159,A 113.6723,B 20.1788,C -0.8011,E1 20.1241,E2 334.3794} C_DIS
LIN {X -56.0914,Y 120.9739,Z 159,A 112.2881,B 20.1785,C -0.8073,E1 20.1275,E2 335.75} C_DIS
LIN {X -53.0314,Y 122.3462,Z 159,A 110.929,B 20.1783,C -0.8126,E1 20.131,E2 337.0978} C_DIS
LIN {X -48.966,Y 124.0312,Z 159,A 108.7518,B 20.1786,C -0.8037,E1 20.1367,E2 339.3072} C_DIS
LIN {X -45.9393,Y 125.1842,Z 159,A 107.4121,B 20.1785,C -0.8074,E1 20.1402,E2 340.6393} C_DIS
LIN {X -43.0264,Y 126.2146,Z 159,A 105.9945,B 20.1785,C -0.8054,E1 20.1439,E2 342.0663} C_DIS
LIN {X -37.0275,Y 128.102,Z 159,A 103.2875,B 20.1785,C -0.8081,E1 20.1512,E2 344.7713} C_DIS
LIN {X -32.9993,Y 129.1977,Z 159,A 101.5178,B 20.1784,C -0.8108,E1 20.1559,E2 346.5367} C_DIS
LIN {X -27.4407,Y 130.4933,Z 159,A 99.0031,B 20.1784,C -0.8103,E1 20.1628,E2 349.0568} C_DIS
LIN {X -24.137,Y 131.1443,Z 159,A 97.5015,B 20.1784,C -0.8091,E1 20.1669,E2 350.5637} C_DIS
LIN {X -19.207,Y 131.9554,Z 159,A 95.5101,B 20.1781,C -0.8168,E1 20.1724,E2 352.5352} C_DIS
LIN {X -16.0505,Y 132.3762,Z 159,A 94.3094,B 20.1778,C -0.8244,E1 20.1756,E2 353.715} C_DIS
LIN {X -12.8534,Y 132.7246,Z 159,A 92.7687,B 20.1781,C -0.8185,E1 20.18,E2 355.2736} C_DIS
LIN {X -8.9147,Y 133.0491,Z 159,A 90.9683,B 20.1781,C -0.815,E1 20.185,E2 357.0852} C_DIS
LIN {X -5.0501,Y 133.25,Z 159,A 89.4241,B 20.178,C -0.8203,E1 20.1893,E2 358.6143} C_DIS
LIN {X -1.1333,Y 133.3414,Z 159,A 87.7219,B 20.178,C -0.8199,E1 20.194,E2 360.318} C_DIS
LIN {X 2.2964,Y 133.3259,Z 159,A 86.2487,B 20.178,C -0.8201,E1 20.1981,E2 361.7904} C_DIS
LIN {X 6.3988,Y 133.1923,Z 159,A 84.4702,B 20.178,C -0.8195,E1 20.2031,E2 363.5699} C_DIS
LIN {X 10.4507,Y 132.9375,Z 159,A 82.6316,B 20.1782,C -0.8155,E1 20.2083,E2 365.4191} C_DIS
LIN {X 14.317,Y 132.5747,Z 159,A 81.0615,B 20.178,C -0.8193,E1 20.2126,E2 366.9769} C_DIS
LIN {X 18.62,Y 132.0392,Z 159,A 79.21,B 20.178,C -0.8193,E1 20.2177,E2 368.8264} C_DIS
LIN {X 22.2409,Y 131.4778,Z 159,A 77.6427,B 20.178,C -0.819,E1 20.222,E2 370.3925} C_DIS
LIN {X 26.2181,Y 130.743,Z 159,A 76.103,B 20.1777,C -0.8265,E1 20.2262,E2 371.9082} C_DIS
LIN {X 28.7826,Y 130.2036,Z 159,A 74.8484,B 20.178,C -0.8205,E1 20.2297,E2 373.178} C_DIS
LIN {X 31.9531,Y 129.4619,Z 159,A 73.2974,B 20.1783,C -0.8133,E1 20.2339,E2 374.7471} C_DIS
LIN {X 35.2837,Y 128.5941,Z 159,A 71.8565,B 20.1783,C -0.8139,E1 20.2378,E2 376.1833} C_DIS
LIN {X 39.8754,Y 127.2456,Z 159,A 69.8944,B 20.1781,C -0.8163,E1 20.243,E2 378.1342} C_DIS
LIN {X 43.4502,Y 126.0677,Z 159,A 68.2646,B 20.1782,C -0.8144,E1 20.2473,E2 379.7654} C_DIS
LIN {X 46.4709,Y 124.9859,Z 159,A 66.863,B 20.1783,C -0.8122,E1 20.251,E2 381.1698} C_DIS
LIN {X 49.6007,Y 123.7771,Z 159,A 65.4235,B 20.1783,C -0.8108,E1 20.2547,E2 382.6093} C_DIS
LIN {X 52.4866,Y 122.5818,Z 159,A 64.0474,B 20.1785,C -0.8079,E1 20.2583,E2 383.9897} C_DIS
LIN {X 55.8255,Y 121.0969,Z 159,A 62.4916,B 20.1785,C -0.8067,E1 20.2623,E2 385.544} C_DIS
LIN {X 58.8321,Y 119.665,Z 159,A 61.1997,B 20.1784,C -0.8108,E1 20.2655,E2 386.8195} C_DIS
LIN {X 61.6547,Y 118.2359,Z 159,A 59.7468,B 20.1786,C -0.805,E1 20.2691,E2 388.2841} C_DIS
LIN {X 65.3465,Y 116.2379,Z 159,A 57.9981,B 20.1786,C -0.8049,E1 20.2734,E2 390.0268} C_DIS
LIN {X 67.7618,Y 114.847,Z 159,A 56.6606,B 20.1789,C -0.7971,E1 20.2766,E2 391.3816} C_DIS
LIN {X 71.5535,Y 112.5242,Z 159,A 54.7614,B 20.1789,C -0.7947,E1 20.2811,E2 393.2801} C_DIS
LIN {X 75.1767,Y 110.1363,Z 159,A 52.8932,B 20.1791,C -0.7915,E1 20.2855,E2 395.1497} C_DIS
LIN {X 78.7873,Y 107.5827,Z 159,A 51.0122,B 20.1791,C -0.789,E1 20.2897,E2 397.0293} C_DIS
LIN {X 82.8222,Y 104.5083,Z 159,A 48.8316,B 20.1793,C -0.785,E1 20.2945,E2 399.2112} C_DIS
LIN {X 86.2758,Y 101.6756,Z 159,A 46.9728,B 20.1793,C -0.784,E1 20.2985,E2 401.064} C_DIS
LIN {X 89.2581,Y 99.0685,Z 159,A 45.2183,B 20.1796,C -0.7783,E1 20.3022,E2 402.826} C_DIS
LIN {X 92.5755,Y 95.9753,Z 159,A 43.2916,B 20.1796,C -0.7753,E1 20.3061,E2 404.7513} C_DIS
LIN {X 95.8341,Y 92.7213,Z 159,A 41.3726,B 20.1798,C -0.7737,E1 20.3098,E2 406.6646} C_DIS
LIN {X 98.921,Y 89.4211,Z 159,A 39.3966,B 20.18,C -0.7679,E1 20.3136,E2 408.6463} C_DIS
LIN {X 101.7846,Y 86.1475,Z 159,A 37.6312,B 20.18,C -0.7681,E1 20.3168,E2 410.4008} C_DIS
LIN {X 104.451,Y 82.8942,Z 159,A 35.764,B 20.1802,C -0.7613,E1 20.3201,E2 412.2769} C_DIS
LIN {X 107.1295,Y 79.4026,Z 159,A 33.8834,B 20.1804,C -0.7571,E1 20.3232,E2 414.1581} C_DIS
LIN {X 109.5079,Y 76.0885,Z 159,A 32.1701,B 20.1804,C -0.7545,E1 20.326,E2 415.8683} C_DIS
LIN {X 111.9846,Y 72.3944,Z 159,A 30.2459,B 20.1806,C -0.749,E1 20.329,E2 417.7961} C_DIS
LIN {X 114.3654,Y 68.5719,Z 159,A 28.3059,B 20.1808,C -0.7438,E1 20.3318,E2 419.7388} C_DIS
LIN {X 116.5008,Y 64.8776,Z 159,A 26.4653,B 20.181,C -0.7386,E1 20.3343,E2 421.5823} C_DIS
LIN {X 118.6756,Y 60.8039,Z 159,A 24.7165,B 20.1808,C -0.7437,E1 20.3366,E2 423.3046} C_DIS
LIN {X 119.9186,Y 58.3181,Z 159,A 23.262,B 20.1814,C -0.7288,E1 20.3384,E2 424.7923} C_DIS
LIN {X 121.6618,Y 54.5833,Z 159,A 21.6839,B 20.1812,C -0.7324,E1 20.3402,E2 426.349} C_DIS
LIN {X 122.8992,Y 51.7384,Z 159,A 20.304,B 20.1814,C -0.7265,E1 20.3417,E2 427.7363} C_DIS
LIN {X 124.1978,Y 48.5374,Z 159,A 18.88,B 20.1814,C -0.725,E1 20.3432,E2 429.1548} C_DIS
LIN {X 125.4015,Y 45.3366,Z 159,A 17.4571,B 20.1816,C -0.7228,E1 20.3446,E2 430.574} C_DIS
LIN {X 126.3405,Y 42.6534,Z 159,A 16.2345,B 20.1816,C -0.7191,E1 20.3457,E2 431.7983} C_DIS
LIN {X 127.7262,Y 38.3084,Z 159,A 14.2373,B 20.1819,C -0.7116,E1 20.3474,E2 433.8028} C_DIS
LIN {X 128.775,Y 34.6127,Z 159,A 12.7793,B 20.1819,C -0.7153,E1 20.3484,E2 435.2394} C_DIS
LIN {X 129.5145,Y 31.7365,Z 159,A 11.2956,B 20.1823,C -0.7021,E1 20.3495,E2 436.7503} C_DIS
LIN {X 130.6579,Y 26.6362,Z 159,A 9.0104,B 20.1825,C -0.6935,E1 20.3508,E2 439.0434} C_DIS
LIN {X 131.4781,Y 22.2395,Z 159,A 7.2565,B 20.1825,C -0.6951,E1 20.3517,E2 440.7796} C_DIS
LIN {X 132.0746,Y 18.3726,Z 159,A 5.4351,B 20.1829,C -0.6836,E1 20.3524,E2 442.6206} C_DIS
LIN {X 132.572,Y 14.3419,Z 159,A 3.8178,B 20.1829,C -0.6839,E1 20.3529,E2 444.2249} C_DIS
LIN {X 132.9369,Y 10.4578,Z 159,A 2.06,B 20.1831,C -0.675,E1 20.3534,E2 445.9953} C_DIS
LIN {X 133.178,Y 6.6825,Z 159,A 0.5248,B 20.1831,C -0.674,E1 20.3536,E2 447.5219} C_DIS
LIN {X 133.3223,Y 2.5086,Z 159,A -1.2237,B 20.1833,C -0.6704,E1 20.3537,E2 449.2676} C_DIS
LIN {X 133.3404,Y -1.3445,Z 159,A -2.8968,B 20.1835,C -0.6643,E1 20.3537,E2 450.9454} C_DIS
LIN {X 133.2237,Y -5.7254,Z 159,A -4.8171,B 20.1837,C -0.6567,E1 20.3536,E2 452.8732} C_DIS
LIN {X 133.0061,Y -9.5099,Z 159,A -6.3522,B 20.1837,C -0.6558,E1 20.3533,E2 454.3993} C_DIS
LIN {X 132.6918,Y -13.1948,Z 159,A -8.0521,B 20.1841,C -0.6458,E1 20.3528,E2 456.1154} C_DIS
LIN {X 132.2441,Y -17.1039,Z 159,A -9.4871,B 20.1839,C -0.652,E1 20.3524,E2 457.5218} C_DIS
LIN {X 131.8802,Y -19.7254,Z 159,A -10.9009,B 20.1844,C -0.6359,E1 20.3518,E2 458.9714} C_DIS
LIN {X 131.0973,Y -24.3911,Z 159,A -12.7148,B 20.1843,C -0.6394,E1 20.3509,E2 460.7617} C_DIS
LIN {X 130.5665,Y -27.0853,Z 159,A -14.1,B 20.1846,C -0.6264,E1 20.3501,E2 462.1739} C_DIS
LIN {X 129.6369,Y -31.2289,Z 159,A -15.7379,B 20.1846,C -0.6292,E1 20.3491,E2 463.792} C_DIS
LIN {X 128.8273,Y -34.4165,Z 159,A -17.1375,B 20.1846,C -0.6254,E1 20.3481,E2 465.1922} C_DIS
LIN {X 127.7292,Y -38.2983,Z 159,A -19.1022,B 20.1851,C -0.6096,E1 20.3466,E2 467.1882} C_DIS
LIN {X 126.1517,Y -43.2079,Z 159,A -21.1121,B 20.1851,C -0.6121,E1 20.3448,E2 469.1764} C_DIS
LIN {X 124.3803,Y -48.0679,Z 159,A -23.141,B 20.1851,C -0.6142,E1 20.3429,E2 471.1851} C_DIS
LIN {X 123.42,Y -50.4865,Z 159,A -24.5218,B 20.1854,C -0.5989,E1 20.3414,E2 472.6} C_DIS
LIN {X 121.9263,Y -53.9919,Z 159,A -26.056,B 20.1854,C -0.5987,E1 20.3397,E2 474.1242} C_DIS
LIN {X 120.4112,Y -57.2895,Z 159,A -27.476,B 20.1854,C -0.6004,E1 20.338,E2 475.5296} C_DIS
LIN {X 119.1994,Y -59.7748,Z 159,A -28.8555,B 20.1857,C -0.5883,E1 20.3363,E2 476.9347} C_DIS
LIN {X 117.2965,Y -63.4278,Z 159,A -30.5931,B 20.1858,C -0.5847,E1 20.334,E2 478.6711} C_DIS
LIN {X 115.1785,Y -67.1975,Z 159,A -32.4037,B 20.1859,C -0.5815,E1 20.3315,E2 480.4789} C_DIS
LIN {X 112.979,Y -70.8332,Z 159,A -34.0745,B 20.1859,C -0.5834,E1 20.3291,E2 482.1336} C_DIS
LIN {X 110.9863,Y -73.9154,Z 159,A -35.5937,B 20.1859,C -0.5817,E1 20.3268,E2 483.6481} C_DIS
LIN {X 108.7004,Y -77.2383,Z 159,A -37.9422,B 20.1868,C -0.5495,E1 20.3229,E2 486.0748} C_DIS
LIN {X 106.0794,Y -80.7999,Z 159,A -39.6562,B 20.1868,C -0.5528,E1 20.32,E2 487.769} C_DIS
LIN {X 103.9031,Y -83.5799,Z 159,A -40.9196,B 20.1865,C -0.5601,E1 20.3179,E2 489.0037} C_DIS
LIN {X 100.9948,Y -87.0717,Z 159,A -42.8494,B 20.1866,C -0.5562,E1 20.3144,E2 490.9337} C_DIS
LIN {X 97.8112,Y -90.6338,Z 159,A -44.9704,B 20.1868,C -0.5481,E1 20.3104,E2 493.0661} C_DIS
LIN {X 94.3339,Y -94.248,Z 159,A -46.9753,B 20.1868,C -0.5496,E1 20.3065,E2 495.0557} C_DIS
LIN {X 91.2968,Y -97.1926,Z 159,A -48.7733,B 20.1868,C -0.5463,E1 20.3028,E2 496.8539} C_DIS
LIN {X 88.5743,Y -99.68,Z 159,A -50.5312,B 20.1872,C -0.535,E1 20.2991,E2 498.6353} C_DIS
LIN {X 84.7067,Y -102.9872,Z 159,A -52.5721,B 20.1872,C -0.5367,E1 20.2948,E2 500.6614} C_DIS
LIN {X 81.3474,Y -105.6608,Z 159,A -54.4658,B 20.1872,C -0.5307,E1 20.2906,E2 502.5636} C_DIS
LIN {X 78.3302,Y -107.9157,Z 159,A -56.2072,B 20.1875,C -0.522,E1 20.2867,E2 504.3221} C_DIS
LIN {X 74.2516,Y -110.7619,Z 159,A -59.3099,B 20.1886,C -0.4759,E1 20.2792,E2 507.5447} C_DIS
LIN {X 67.2759,Y -115.1324,Z 159,A -61.6888,B 20.1875,C -0.5198,E1 20.2738,E2 509.7876} C_DIS
LIN {X 63.4714,Y -117.2731,Z 159,A -63.3763,B 20.1875,C -0.5249,E1 20.2697,E2 511.4542} C_DIS
LIN {X 61.0358,Y -118.5576,Z 159,A -64.538,B 20.1875,C -0.5239,E1 20.2669,E2 512.6146} C_DIS
LIN {X 58.5886,Y -119.7851,Z 159,A -65.9491,B 20.1877,C -0.5118,E1 20.2633,E2 514.0558} C_DIS
LIN {X 54.6113,Y -121.6493,Z 159,A -67.6502,B 20.1877,C -0.5171,E1 20.259,E2 515.7361} C_DIS
Enddeposition()
END
